ABB RobotStudio station: P4.rspag

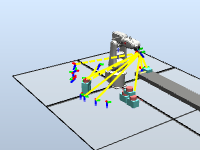
--- station ---
Station CPRClasificador (saved by RobotStudio 6.6.7701.1025)
Controller IRB_120_3kg_0.58m_1
  mechanical unit ROB_1: IRB120_3_58__01, 6 joints, base frame (0, 0, 0) mm
Layout (positions relative to the parent item):
  - Cinta [part]
  - Placa [part]
  - Disco [part]
  - CI_Ventosa [smart component]
      signals: DI ActivaVentosa, DO Vacuostato
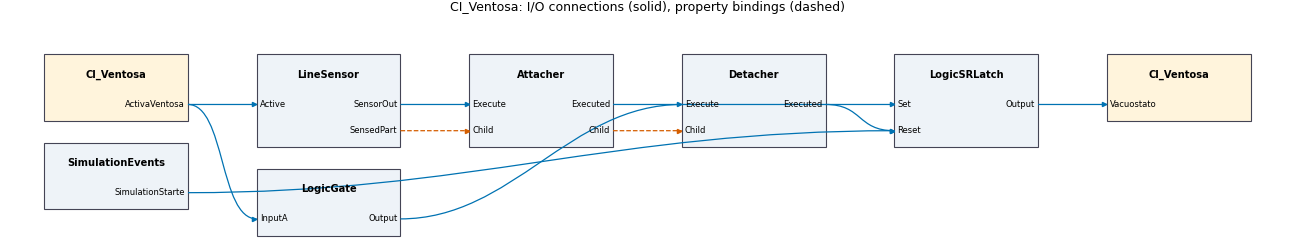
      connections:
        CI_Ventosa.ActivaVentosa -> LineSensor.Active
        LineSensor.SensorOut -> Attacher.Execute
        Attacher.Executed -> LogicSRLatch.Set
        Detacher.Executed -> LogicSRLatch.Reset
        CI_Ventosa.ActivaVentosa -> LogicGate.InputA
        LogicSRLatch.Output -> CI_Ventosa.Vacuostato
        SimulationEvents.SimulationStarted -> LogicSRLatch.Reset
        LogicGate.Output -> Detacher.Execute
        LineSensor.SensedPart => Attacher.Child
        Attacher.Child => Detacher.Child
    - LineSensor [smart component, from Components\LineSensor.rslib] at (364.35, 0, 594) mm, rotated rx 180 ry 60 rz 180 deg
        properties: Start=[0 0 0.049]; End=[0 0 0.061]; Radius=0.002; SensedPart=Disco_79; SensedPoint=[0.464333557128906 -0.180395202636719 0.20952131652832]
      - _sensorPart_ [part]
    - Attacher [smart component, from Components\Attacher.rslib]
        properties: Parent=MyNewTool; Flange=0; Child=Disco_79; Mount=false; Offset=[0 0 0]; Orientation=[0 0 0]
    - Detacher [smart component, from Components\Detacher.rslib]
        properties: Child=Disco_79; KeepPosition=true
    - LogicGate [smart component, from Components\LogicGate.rslib]
        properties: Operator=NOT; Delay=0
    - LogicSRLatch [smart component, from Components\LogicSRLatch.rslib]
    - SimulationEvents [smart component, from Components\SimulationEvents.rslib]
    - MyNewTool [mechanism] at (364.35, 0, 594) mm, rotated rx 180 ry 60 rz 180 deg
        TCP MyNewTool at (0, 0, 50) mm
        links: Cono
  - CI_Cinta [smart component]
      signals: DI ActivaSensores, DO SensorCinta1, DO SensorCinta2
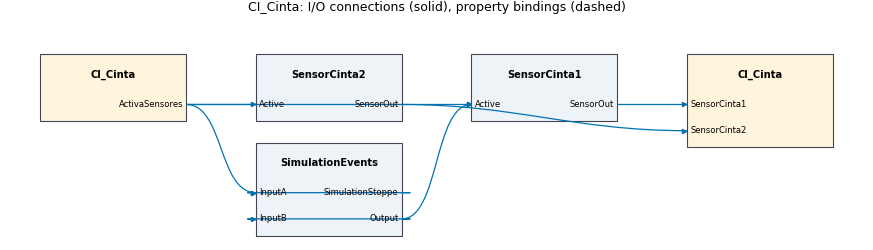
      connections:
        CI_Cinta.ActivaSensores -> SensorCinta2.Active
        SensorCinta1.SensorOut -> CI_Cinta.SensorCinta1
        SensorCinta2.SensorOut -> CI_Cinta.SensorCinta2
        SimulationEvents.SimulationStopped -> LogicGate_2.InputA
        LogicGate_2.Output -> LogicGate.InputB
        CI_Cinta.ActivaSensores -> LogicGate.InputA
        LogicGate.Output -> SensorCinta1.Active
        CI_Cinta.ActivaSensores -> SensorCinta1.Active
    - SensorCinta1 [smart component, from Components\LineSensor.rslib]
        properties: Start=[0.15 0.15 0.22]; End=[0.15 0.35 0.22]; Radius=0.002; SensedPart=Placa_91; SensedPoint=[0.15 0.25 0.22]
      - _sensorPart_ [part]
    - SensorCinta2 [smart component, from Components\LineSensor.rslib]
        properties: Start=[0.25 0.15 0.22]; End=[0.25 0.35 0.22]; Radius=0.002; SensedPart=Placa_91; SensedPoint=[0.25 0.25 0.22]
      - _sensorPart_ [part]
  - CI_Piezas [smart component]
      signals: DI Pieza, DI MotorCinta, DI Desencolar
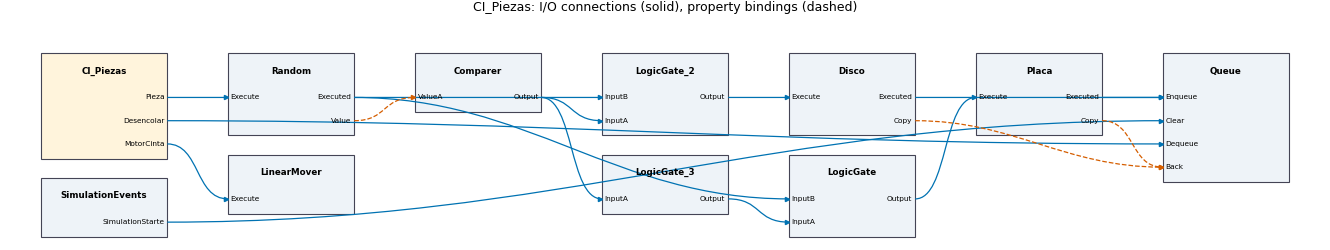
      connections:
        Random.Executed -> LogicGate_2.InputB
        Random.Executed -> LogicGate.InputB
        Comparer.Output -> LogicGate_2.InputA
        Comparer.Output -> LogicGate_3.InputA
        LogicGate_3.Output -> LogicGate.InputA
        LogicGate_2.Output -> Disco.Execute
        Disco.Executed -> Queue.Enqueue
        CI_Piezas.Pieza -> Random.Execute
        SimulationEvents.SimulationStarted -> Queue.Clear
        CI_Piezas.Desencolar -> Queue.Dequeue
        Placa.Executed -> Queue.Enqueue
        LogicGate.Output -> Placa.Execute
        CI_Piezas.MotorCinta -> LinearMover.Execute
        Random.Value => Comparer.ValueA
        Disco.Copy => Queue.Back
        Placa.Copy => Queue.Back
    - Disco [smart component, from Components\Source.rslib]
        properties: Source=Disco; Copy=Disco_171; Parent=(none); Position=[1.25 0.23 0.2]; Orientation=[0 0 0]; Transient=false; PhysicsBehavior=0
    - Random [smart component, from Components\Random.rslib]
        properties: Value=0.259914413215553; Min=0; Max=1
    - Comparer [smart component, from Components\Comparer.rslib]
        properties: ValueA=0.259914413215553; Operator=<=; ValueB=0.5
    - LogicGate [smart component, from Components\LogicGate.rslib]
        properties: Operator=AND; Delay=0
    - LogicGate_2 [smart component, from Components\LogicGate.rslib]
        properties: Operator=AND; Delay=0
    - LogicGate_3 [smart component, from Components\LogicGate.rslib]
        properties: Operator=NOT; Delay=0
    - LinearMover [smart component, from Components\LinearMover.rslib]
        properties: Object=Queue; Direction=[-1 0 0]; Speed=0.15; Reference=Global; ReferenceObject=(none)
    - SimulationEvents [smart component, from Components\SimulationEvents.rslib]
    - Queue [smart component, from Components\Queue.rslib]
        properties: Back=Disco_171; Front=Disco_171; Queue={b508ca64-a9cf-4086-8e21-28a4116258de}; NumberOfObjects=1
    - Placa [smart component, from Components\Source.rslib]
        properties: Source=Placa; Copy=Placa_170; Parent=(none); Position=[1.15 0.25 0.2]; Orientation=[0 0 0]; Transient=false; PhysicsBehavior=0
  - IRB120_3_58__01 [mechanism, from Robots\IRB120_3_58_G_01.rslib] at (0, 0, 0) mm; joint values [0, 0, 0, 0, 0.5236, 0] (rad or m)
  - Placa_75 [part] at (1150, 250, 200) mm
  - Placa_81 [part] at (1150, 250, 200) mm
  - Placa_83 [part] at (1150, 250, 200) mm
  - Placa_84 [part] at (1150, 250, 200) mm
  - Placa_85 [part] at (1150, 250, 200) mm
  - Placa_86 [part] at (1150, 250, 200) mm
  - Placa_88 [part] at (1150, 250, 200) mm
  - Placa_93 [part] at (1150, 250, 200) mm
  - Placa_94 [part] at (1150, 250, 200) mm
  - Placa_95 [part] at (1150, 250, 200) mm
  - Placa_97 [part] at (1150, 250, 200) mm
  - Placa_99 [part] at (1150, 250, 200) mm
  - Placa_101 [part] at (1150, 250, 200) mm
  - Placa_102 [part] at (1150, 250, 200) mm
  - Placa_103 [part] at (1150, 250, 200) mm
  - Placa_104 [part] at (1150, 250, 200) mm
  - Disco_105 [part] at (1250, 230, 200) mm
  - Disco_106 [part] at (1250, 230, 200) mm
  - Disco_107 [part] at (1250, 230, 200) mm
  - Disco_108 [part] at (1250, 230, 200) mm
  - Placa_110 [part] at (1150, 250, 200) mm
  - Placa_111 [part] at (1150, 250, 200) mm
  - Placa_113 [part] at (1150, 250, 200) mm
  - Disco_114 [part] at (1250, 230, 200) mm
  - Disco_115 [part] at (1250, 230, 200) mm
  - Placa_116 [part] at (1150, 250, 200) mm
  - Placa_117 [part] at (1150, 250, 200) mm
  - Disco_118 [part] at (1250, 230, 200) mm
  - Placa_119 [part] at (1150, 250, 200) mm
  - Disco_120 [part] at (1250, 230, 200) mm
  - Disco_121 [part] at (1250, 230, 200) mm
  - Disco_122 [part] at (1250, 230, 200) mm
  - Disco_123 [part] at (1250, 230, 200) mm
  - Placa_124 [part] at (1150, 250, 200) mm
  - Placa_125 [part] at (1150, 250, 200) mm
  - Placa_126 [part] at (1150, 250, 200) mm
  - Disco_127 [part] at (1250, 230, 200) mm
  - Placa_128 [part] at (1150, 250, 200) mm
  - Disco_129 [part] at (1250, 230, 200) mm
  - Placa_130 [part] at (1150, 250, 200) mm
  - Disco_131 [part] at (1250, 230, 200) mm
  - Placa_132 [part] at (1150, 250, 200) mm
  - Placa_133 [part] at (1150, 250, 200) mm
  - Placa_134 [part] at (1150, 250, 200) mm
  - Disco_135 [part] at (1250, 230, 200) mm
  - Disco_137 [part] at (1250, 230, 200) mm
  - Disco_138 [part] at (1250, 230, 200) mm
  - Disco_139 [part] at (1250, 230, 200) mm
  - Disco_140 [part] at (1250, 230, 200) mm
  - Disco_141 [part] at (1250, 230, 200) mm
  - Disco_142 [part] at (1250, 230, 200) mm
  - Placa_143 [part] at (1150, 250, 200) mm
  - Placa_144 [part] at (1150, 250, 200) mm
  - Disco_145 [part] at (1250, 230, 200) mm
  - Placa_146 [part] at (1150, 250, 200) mm
  - Disco_147 [part] at (1250, 230, 200) mm
  - Disco_148 [part] at (1250, 230, 200) mm
  - Placa_149 [part] at (1150, 250, 200) mm
  - Placa_150 [part] at (1150, 250, 200) mm
  - Disco_151 [part] at (1250, 230, 200) mm
  - Disco_152 [part] at (1250, 230, 200) mm
  - Placa_153 [part] at (1150, 250, 200) mm
  - Disco_154 [part] at (1250, 230, 200) mm
  - Placa_155 [part] at (1150, 250, 200) mm
  - Placa_156 [part] at (1150, 250, 200) mm
  - Disco_157 [part] at (1250, 230, 200) mm
  - Disco_158 [part] at (1250, 230, 200) mm
  - Placa_159 [part] at (1150, 250, 200) mm
  - Placa_161 [part] at (1150, 250, 200) mm
  - Placa_162 [part] at (1150, 250, 200) mm
  - Placa_163 [part] at (1150, 250, 200) mm
  - Disco_164 [part] at (1250, 230, 200) mm
  - Disco_165 [part] at (1250, 230, 200) mm
  - Placa_166 [part] at (1150, 250, 200) mm
  - Placa_167 [part] at (1150, 250, 200) mm
  - Disco_168 [part] at (1250, 230, 200) mm
  - Placa_169 [part] at (1150, 250, 200) mm
  - Disco_170 [part] at (1250, 230, 200) mm
  - Disco_171 [part] at (1250, 230, 200) mm
  - Disco_172 [part] at (1250, 230, 200) mm
  - Disco_173 [part] at (1250, 230, 200) mm
  - Disco_174 [part] at (1250, 230, 200) mm
  - Disco_175 [part] at (1250, 230, 200) mm
  - Disco_176 [part] at (1250, 230, 200) mm
  - Disco_177 [part] at (1250, 230, 200) mm
  - Disco_178 [part] at (1250, 230, 200) mm
  - Disco_179 [part] at (1250, 230, 200) mm
  - Disco_180 [part] at (1250, 230, 200) mm
  - Disco_181 [part] at (1250, 230, 200) mm
  - Placa_182 [part] at (1150, 250, 200) mm
  - Disco_183 [part] at (1250, 230, 200) mm
  - Disco_185 [part] at (1250, 230, 200) mm
  - Placa_186 [part] at (1150, 250, 200) mm
  - Disco_187 [part] at (1250, 230, 200) mm
  - Disco_188 [part] at (1250, 230, 200) mm
  - Placa_189 [part] at (1150, 250, 200) mm
  - Placa_190 [part] at (1150, 250, 200) mm
  - Placa_191 [part] at (1150, 250, 200) mm
  - Disco_192 [part] at (1250, 230, 200) mm
  - Disco_193 [part] at (1250, 230, 200) mm
  - Placa_194 [part] at (1150, 250, 200) mm
  - Disco_195 [part] at (1250, 230, 200) mm
  - Placa_196 [part] at (1150, 250, 200) mm
  - Placa_197 [part] at (1150, 250, 200) mm
  - Disco_198 [part] at (1250, 230, 200) mm
  - Disco_199 [part] at (1250, 230, 200) mm
  - Placa_200 [part] at (1150, 250, 200) mm
  - Placa_201 [part] at (1150, 250, 200) mm
  - Disco_202 [part] at (1250, 230, 200) mm
  - Placa_203 [part] at (1150, 250, 200) mm
  - Disco_204 [part] at (1250, 230, 200) mm
  - Disco_205 [part] at (1250, 230, 200) mm
  - Disco_206 [part] at (1250, 230, 200) mm
  - Disco_207 [part] at (1250, 230, 200) mm
  - Disco_209 [part] at (1250, 230, 200) mm
  - Placa_210 [part] at (1150, 250, 200) mm
  - Disco_211 [part] at (1250, 230, 200) mm
  - Disco_212 [part] at (1250, 230, 200) mm
  - Placa_213 [part] at (1150, 250, 200) mm
  - Placa_214 [part] at (1150, 250, 200) mm
  - Placa_215 [part] at (1150, 250, 200) mm
  - Disco_216 [part] at (1250, 230, 200) mm
  - Placa_217 [part] at (1150, 250, 200) mm
  - Disco_218 [part] at (1250, 230, 200) mm
  - Disco_219 [part] at (1250, 230, 200) mm
  - Disco_220 [part] at (1250, 230, 200) mm
  - Placa_221 [part] at (1150, 250, 200) mm
  - Placa_222 [part] at (1150, 250, 200) mm
  - Placa_223 [part] at (1150, 250, 200) mm
  - Disco_224 [part] at (1250, 230, 200) mm
  - Placa_225 [part] at (1150, 250, 200) mm
  - Disco_226 [part] at (1250, 230, 200) mm
  - Placa_227 [part] at (1150, 250, 200) mm
  - Placa_228 [part] at (1150, 250, 200) mm
  - Placa_229 [part] at (1150, 250, 200) mm
  - Placa_230 [part] at (1150, 250, 200) mm
  - Disco_231 [part] at (1250, 230, 200) mm
  - Placa_232 [part] at (1150, 250, 200) mm
  - Disco_233 [part] at (1250, 230, 200) mm
  - Placa_234 [part] at (1150, 250, 200) mm
  - Disco_235 [part] at (1250, 230, 200) mm
  - Disco_236 [part] at (1250, 230, 200) mm
  - Disco_237 [part] at (1250, 230, 200) mm
  - Placa_238 [part] at (1150, 250, 200) mm
  - Disco_239 [part] at (1250, 230, 200) mm
  - Disco_240 [part] at (1250, 230, 200) mm
  - Disco_241 [part] at (1250, 230, 200) mm
  - Placa_242 [part] at (1150, 250, 200) mm
  - Placa_243 [part] at (1150, 250, 200) mm
  - Placa_244 [part] at (1150, 250, 200) mm
  - Disco_245 [part] at (1250, 230, 200) mm
  - Placa_246 [part] at (1150, 250, 200) mm
  - Disco_247 [part] at (1250, 230, 200) mm
  - Placa_248 [part] at (1150, 250, 200) mm
  - Placa_249 [part] at (1150, 250, 200) mm
  - Disco_250 [part] at (1250, 230, 200) mm
  - Disco_251 [part] at (1250, 230, 200) mm
  - Disco_252 [part] at (1250, 230, 200) mm
  - Disco_253 [part] at (1250, 230, 200) mm
  - Placa_254 [part] at (1150, 250, 200) mm
  - Disco_255 [part] at (1250, 230, 200) mm
  - Placa_256 [part] at (1150, 250, 200) mm
  - Disco_257 [part] at (1250, 230, 200) mm
  - Placa_258 [part] at (1150, 250, 200) mm
  - Placa_259 [part] at (1150, 250, 200) mm
  - Disco_260 [part] at (1250, 230, 200) mm
  - Disco_261 [part] at (1250, 230, 200) mm
  - Placa_262 [part] at (1150, 250, 200) mm
  - Placa_263 [part] at (1150, 250, 200) mm
  - Placa_264 [part] at (1150, 250, 200) mm
  - Disco_265 [part] at (1250, 230, 200) mm
  - Disco_266 [part] at (1250, 230, 200) mm
  - Placa_267 [part] at (1150, 250, 200) mm
  - Disco_268 [part] at (1250, 230, 200) mm
  - Disco_269 [part] at (1250, 230, 200) mm
  - Disco_270 [part] at (1250, 230, 200) mm
  - Placa_271 [part] at (1150, 250, 200) mm
  - Placa_272 [part] at (1150, 250, 200) mm
  - Disco_273 [part] at (1250, 230, 200) mm
  - Disco_274 [part] at (1250, 230, 200) mm
  - Placa_275 [part] at (1150, 250, 200) mm
  - Placa_276 [part] at (1150, 250, 200) mm
  - Disco_277 [part] at (1250, 230, 200) mm
  - Placa_278 [part] at (1150, 250, 200) mm
  - Placa_279 [part] at (1150, 250, 200) mm
  - Disco_280 [part] at (1250, 230, 200) mm
  - Placa_281 [part] at (1150, 250, 200) mm
  - Disco_282 [part] at (1250, 230, 200) mm
  - Placa_283 [part] at (1150, 250, 200) mm
  - Disco_284 [part] at (1250, 230, 200) mm
  - Disco_285 [part] at (1250, 230, 200) mm
  - Disco_286 [part] at (1250, 230, 200) mm
  - Placa_287 [part] at (1150, 250, 200) mm
  - Disco_288 [part] at (1250, 230, 200) mm
  - Disco_289 [part] at (1250, 230, 200) mm
  - Disco_290 [part] at (1250, 230, 200) mm
  - Placa_291 [part] at (1150, 250, 200) mm
  - Placa_292 [part] at (1150, 250, 200) mm
  - Placa_293 [part] at (1150, 250, 200) mm
  - Placa_294 [part] at (1150, 250, 200) mm
  - Placa_295 [part] at (1150, 250, 200) mm
  - Placa_296 [part] at (1150, 250, 200) mm
  - Placa_297 [part] at (1150, 250, 200) mm
  - Placa_298 [part] at (1150, 250, 200) mm
  - Disco_299 [part] at (1250, 230, 200) mm
  - Placa_300 [part] at (1150, 250, 200) mm
  - Placa_301 [part] at (1150, 250, 200) mm
  - Disco_302 [part] at (1250, 230, 200) mm
  - Disco_303 [part] at (1250, 230, 200) mm
  - Placa_304 [part] at (1150, 250, 200) mm
  - Placa_305 [part] at (1150, 250, 200) mm
  - Disco_306 [part] at (1250, 230, 200) mm
  - Disco_307 [part] at (1250, 230, 200) mm
  - Placa_308 [part] at (1150, 250, 200) mm
  - Placa_309 [part] at (1150, 250, 200) mm
  - Disco_310 [part] at (1250, 230, 200) mm
  - Placa_311 [part] at (1150, 250, 200) mm
  - Placa_312 [part] at (1150, 250, 200) mm
  - Placa_313 [part] at (1150, 250, 200) mm
  - Placa_314 [part] at (1150, 250, 200) mm
  - Placa_315 [part] at (1150, 250, 200) mm
  - Placa_316 [part] at (1150, 250, 200) mm
  - Disco_317 [part] at (1250, 230, 200) mm
  - Placa_318 [part] at (1150, 250, 200) mm
  - Disco_319 [part] at (1250, 230, 200) mm
  - Disco_320 [part] at (1250, 230, 200) mm
  - Placa_321 [part] at (1150, 250, 200) mm
  - Placa_322 [part] at (1150, 250, 200) mm
  - Placa_323 [part] at (1150, 250, 200) mm
  - Disco_324 [part] at (1250, 230, 200) mm
  - Disco_325 [part] at (1250, 230, 200) mm
  - Disco_326 [part] at (1250, 230, 200) mm
  - Placa_327 [part] at (1150, 250, 200) mm
  - Disco_328 [part] at (1250, 230, 200) mm
  - Disco_329 [part] at (1250, 230, 200) mm
  - Disco_330 [part] at (1250, 230, 200) mm
  - Disco_331 [part] at (1250, 230, 200) mm
  - Disco_332 [part] at (1250, 230, 200) mm
  - Disco_333 [part] at (1250, 230, 200) mm
  - Placa_334 [part] at (1150, 250, 200) mm
  - Disco_335 [part] at (1250, 230, 200) mm
  - Placa_336 [part] at (1150, 250, 200) mm
  - Disco_337 [part] at (1250, 230, 200) mm
  - Placa_338 [part] at (1150, 250, 200) mm
  - Placa_339 [part] at (1150, 250, 200) mm
  - Disco_340 [part] at (1250, 230, 200) mm
  - Placa_341 [part] at (1150, 250, 200) mm
  - Disco_342 [part] at (1250, 230, 200) mm
  - Disco_343 [part] at (1250, 230, 200) mm
  - Disco_344 [part] at (1250, 230, 200) mm
  - Disco_345 [part] at (1250, 230, 200) mm
  - Disco_346 [part] at (1250, 230, 200) mm
  - Placa_347 [part] at (1150, 250, 200) mm
  - Disco_348 [part] at (1250, 230, 200) mm
  - Disco_349 [part] at (1250, 230, 200) mm
  - Disco_350 [part] at (1250, 230, 200) mm
  - Placa_351 [part] at (1150, 250, 200) mm
  - Disco_7 [part] at (1250, 230, 200) mm
  - Disco_8 [part] at (1250, 230, 200) mm
  - Disco_9 [part] at (1250, 230, 200) mm
  - Disco_10 [part] at (1250, 230, 200) mm
  - Disco_11 [part] at (1250, 230, 200) mm
  - Disco_12 [part] at (1250, 230, 200) mm
  - Disco_13 [part] at (1250, 230, 200) mm
  - Disco_14 [part] at (1250, 230, 200) mm
  - Placa_15 [part] at (1150, 250, 200) mm
  - Placa_16 [part] at (1150, 250, 200) mm
  - Placa_17 [part] at (1150, 250, 200) mm
  - Disco_18 [part] at (1250, 230, 200) mm
  - Disco_20 [part] at (1250, 230, 200) mm
  - Placa_21 [part] at (1150, 250, 200) mm
  - Placa_22 [part] at (1150, 250, 200) mm
  - Placa_23 [part] at (1150, 250, 200) mm
  - Disco_24 [part] at (1250, 230, 200) mm
  - Disco_25 [part] at (1250, 230, 200) mm
  - Placa_26 [part] at (1150, 250, 200) mm
  - Placa_27 [part] at (1150, 250, 200) mm
  - Disco_28 [part] at (1250, 230, 200) mm
  - Disco_29 [part] at (1250, 230, 200) mm
  - Placa_30 [part] at (1150, 250, 200) mm
  - Placa_31 [part] at (1150, 250, 200) mm
  - Placa_32 [part] at (1150, 250, 200) mm
  - Disco_33 [part] at (1250, 230, 200) mm
  - Disco_34 [part] at (1250, 230, 200) mm
  - Placa_35 [part] at (1150, 250, 200) mm
  - Placa_36 [part] at (1150, 250, 200) mm
  - Placa_37 [part] at (1150, 250, 200) mm
  - Disco_38 [part] at (1250, 230, 200) mm
  - Disco_39 [part] at (1250, 230, 200) mm
  - Placa_40 [part] at (1150, 250, 200) mm
  - Placa_41 [part] at (1150, 250, 200) mm
  - Placa_42 [part] at (1150, 250, 200) mm
  - Placa_44 [part] at (1150, 250, 200) mm
  - Placa_45 [part] at (1150, 250, 200) mm
  - Disco_46 [part] at (1250, 230, 200) mm
  - Placa_47 [part] at (1150, 250, 200) mm
  - Disco_48 [part] at (1250, 230, 200) mm
  - Placa_49 [part] at (1150, 250, 200) mm
  - Placa_50 [part] at (1150, 250, 200) mm
  - Placa_51 [part] at (1150, 250, 200) mm
  - Disco_52 [part] at (1250, 230, 200) mm
  - Disco_53 [part] at (1250, 230, 200) mm
  - Placa_54 [part] at (1150, 250, 200) mm
  - Placa_55 [part] at (1150, 250, 200) mm
  - Placa_56 [part] at (1150, 250, 200) mm
  - Disco_57 [part] at (1250, 230, 200) mm
  - Disco_58 [part] at (1250, 230, 200) mm
  - Placa_59 [part] at (1150, 250, 200) mm
  - Disco_60 [part] at (1250, 230, 200) mm
  - Disco_61 [part] at (1250, 230, 200) mm
  - Placa_62 [part] at (1150, 250, 200) mm
  - Disco_63 [part] at (1250, 230, 200) mm
  - Disco_64 [part] at (1250, 230, 200) mm
  - Placa_65 [part] at (1150, 250, 200) mm
  - Placa_66 [part] at (1150, 250, 200) mm
  - Disco_68 [part] at (1250, 230, 200) mm
  - Disco_69 [part] at (1250, 230, 200) mm
  - Placa_70 [part] at (1150, 250, 200) mm
  - Disco_71 [part] at (1250, 230, 200) mm
  - Disco_72 [part] at (1250, 230, 200) mm
  - Disco_73 [part] at (1250, 230, 200) mm
  - Disco_74 [part] at (1250, 230, 200) mm
  - Placa_75 [part] at (1150, 250, 200) mm
  - Placa_76 [part] at (1150, 250, 200) mm
  - Disco_77 [part] at (1250, 230, 200) mm
  - Disco_78 [part] at (1250, 230, 200) mm
  - Placa_79 [part] at (1150, 250, 200) mm
  - Placa_80 [part] at (1150, 250, 200) mm
  - Placa_81 [part] at (1150, 250, 200) mm
  - Placa_82 [part] at (1150, 250, 200) mm
  - Disco_83 [part] at (1250, 230, 200) mm
  - Disco_84 [part] at (1250, 230, 200) mm
  - Disco_85 [part] at (1250, 230, 200) mm
  - Placa_86 [part] at (1150, 250, 200) mm
  - Disco_87 [part] at (1250, 230, 200) mm
  - Disco_88 [part] at (1250, 230, 200) mm
  - Disco_89 [part] at (1250, 230, 200) mm
  - Disco_90 [part] at (1250, 230, 200) mm
  - Placa_91 [part] at (1150, 250, 200) mm
  - Disco_92 [part] at (1250, 230, 200) mm
  - Placa_93 [part] at (1150, 250, 200) mm
  - Disco_94 [part] at (1250, 230, 200) mm
  - Placa_95 [part] at (1150, 250, 200) mm
  - Placa_96 [part] at (1150, 250, 200) mm
  - Placa_97 [part] at (1150, 250, 200) mm
  - Disco_98 [part] at (1250, 230, 200) mm
  - Placa_99 [part] at (1150, 250, 200) mm
  - Placa_100 [part] at (1150, 250, 200) mm
  - Disco_101 [part] at (1250, 230, 200) mm
  - Placa_102 [part] at (1150, 250, 200) mm
  - Placa_103 [part] at (1150, 250, 200) mm
  - Disco_104 [part] at (1250, 230, 200) mm
  - Disco_105 [part] at (1250, 230, 200) mm
  - Disco_106 [part] at (1250, 230, 200) mm
  - Disco_107 [part] at (1250, 230, 200) mm
  - Disco_108 [part] at (1250, 230, 200) mm
  - Disco_109 [part] at (1250, 230, 200) mm
  - Placa_110 [part] at (1150, 250, 200) mm
  - Placa_111 [part] at (1150, 250, 200) mm
  - Placa_112 [part] at (1150, 250, 200) mm
  - Disco_113 [part] at (1250, 230, 200) mm
  - Placa_114 [part] at (1150, 250, 200) mm
  - Disco_115 [part] at (1250, 230, 200) mm
  - Disco_116 [part] at (1250, 230, 200) mm
  - Placa_117 [part] at (1150, 250, 200) mm
  - Placa_118 [part] at (1150, 250, 200) mm
  - Disco_119 [part] at (1250, 230, 200) mm
  - Disco_120 [part] at (1250, 230, 200) mm
  - Disco_121 [part] at (1250, 230, 200) mm
  - Placa_122 [part] at (1150, 250, 200) mm
  - Placa_123 [part] at (1150, 250, 200) mm
  - Disco_124 [part] at (1250, 230, 200) mm
  - Placa_125 [part] at (1150, 250, 200) mm
  - Disco_126 [part] at (1250, 230, 200) mm
  - Placa_127 [part] at (1150, 250, 200) mm
  - Placa_128 [part] at (1150, 250, 200) mm
  - Disco_129 [part] at (1250, 230, 200) mm
  - Placa_130 [part] at (1150, 250, 200) mm
  - Disco_131 [part] at (1250, 230, 200) mm
  - Placa_132 [part] at (1150, 250, 200) mm
  - Disco_133 [part] at (1250, 230, 200) mm
  - Disco_134 [part] at (1250, 230, 200) mm
  - Placa_135 [part] at (1150, 250, 200) mm
  - Placa_136 [part] at (1150, 250, 200) mm
  - Disco_137 [part] at (1250, 230, 200) mm
  - Disco_138 [part] at (1250, 230, 200) mm
  - Disco_139 [part] at (1250, 230, 200) mm
  - Placa_140 [part] at (1150, 250, 200) mm
  - Disco_141 [part] at (1250, 230, 200) mm
  - Disco_142 [part] at (1250, 230, 200) mm
  - Placa_143 [part] at (1150, 250, 200) mm
  - Placa_144 [part] at (1150, 250, 200) mm
  - Placa_145 [part] at (1150, 250, 200) mm
  - Placa_146 [part] at (1150, 250, 200) mm
  - Disco_147 [part] at (1250, 230, 200) mm
  - Placa_148 [part] at (1150, 250, 200) mm
  - Placa_149 [part] at (1150, 250, 200) mm
  - Placa_150 [part] at (1150, 250, 200) mm
  - Disco_151 [part] at (1250, 230, 200) mm
  - Disco_152 [part] at (1250, 230, 200) mm
  - Disco_153 [part] at (1250, 230, 200) mm
  - Disco_154 [part] at (1250, 230, 200) mm
  - Disco_155 [part] at (1250, 230, 200) mm
  - Disco_156 [part] at (1250, 230, 200) mm
  - Disco_157 [part] at (1250, 230, 200) mm
  - Disco_158 [part] at (1250, 230, 200) mm
  - Disco_159 [part] at (1250, 230, 200) mm
  - Disco_160 [part] at (1250, 230, 200) mm
  - Placa_161 [part] at (1150, 250, 200) mm
  - Placa_163 [part] at (1150, 250, 200) mm
  - Disco_164 [part] at (1250, 230, 200) mm
  - Placa_165 [part] at (1150, 250, 200) mm
  - Placa_166 [part] at (1150, 250, 200) mm
  - Disco_167 [part] at (1250, 230, 200) mm
  - Disco_168 [part] at (1250, 230, 200) mm
  - Disco_169 [part] at (1250, 230, 200) mm
  - Placa_170 [part] at (1150, 250, 200) mm
  - Disco_171 [part] at (1250, 230, 200) mm
  - Disco_172 [part] at (1250, 230, 200) mm
  - Placa_173 [part] at (1150, 250, 200) mm
  - Disco_174 [part] at (1250, 230, 200) mm
  - Placa_175 [part] at (1150, 250, 200) mm
  - Placa_176 [part] at (1150, 250, 200) mm
  - Disco_177 [part] at (1250, 230, 200) mm
  - Disco_178 [part] at (1250, 230, 200) mm
  - Placa_179 [part] at (1150, 250, 200) mm
  - Placa_180 [part] at (1150, 250, 200) mm
  - Placa_181 [part] at (1150, 250, 200) mm
  - Placa_182 [part] at (1150, 250, 200) mm
  - Disco_183 [part] at (1250, 230, 200) mm
  - Placa_184 [part] at (1150, 250, 200) mm
  - Placa_185 [part] at (1150, 250, 200) mm
  - Disco_186 [part] at (1250, 230, 200) mm
  - Disco_187 [part] at (1250, 230, 200) mm
  - Disco_188 [part] at (1250, 230, 200) mm
  - Placa_189 [part] at (1150, 250, 200) mm
  - Disco_190 [part] at (1250, 230, 200) mm
  - Disco_191 [part] at (1250, 230, 200) mm
  - Placa_192 [part] at (1150, 250, 200) mm
  - Disco_193 [part] at (1250, 230, 200) mm
  - Placa_194 [part] at (1150, 250, 200) mm
  - Disco_195 [part] at (1250, 230, 200) mm
  - Disco_196 [part] at (1250, 230, 200) mm
  - Placa_197 [part] at (1150, 250, 200) mm
  - Disco_198 [part] at (1250, 230, 200) mm
  - Disco_199 [part] at (1250, 230, 200) mm
  - Placa_200 [part] at (1150, 250, 200) mm
  - Disco_201 [part] at (1250, 230, 200) mm
  - Disco_202 [part] at (1250, 230, 200) mm
  - Placa_203 [part] at (1150, 250, 200) mm
  - Placa_204 [part] at (1150, 250, 200) mm
  - Placa_205 [part] at (1150, 250, 200) mm
  - Placa_206 [part] at (1150, 250, 200) mm
  - Disco_207 [part] at (1250, 230, 200) mm
  - Placa_208 [part] at (1150, 250, 200) mm
  - Disco_209 [part] at (1250, 230, 200) mm
  - Placa_219 [part] at (1150, 250, 200) mm
  - Disco_220 [part] at (1250, 230, 200) mm
  - Disco_221 [part] at (1250, 230, 200) mm
  - Disco_222 [part] at (1250, 230, 200) mm
  - Disco_223 [part] at (1250, 230, 200) mm
  - Disco_224 [part] at (1250, 230, 200) mm
  - Placa_225 [part] at (1150, 250, 200) mm
  - Disco_226 [part] at (1250, 230, 200) mm
  - Disco_227 [part] at (1250, 230, 200) mm
  - Placa_228 [part] at (1150, 250, 200) mm
  - Disco_229 [part] at (1250, 230, 200) mm
  - Disco_231 [part] at (1250, 230, 200) mm
  - Placa_232 [part] at (1150, 250, 200) mm
  - Disco_233 [part] at (1250, 230, 200) mm
  - Placa_234 [part] at (1150, 250, 200) mm
  - Placa_235 [part] at (1150, 250, 200) mm
  - Placa_236 [part] at (1150, 250, 200) mm
  - Disco_237 [part] at (1250, 230, 200) mm
  - Placa_238 [part] at (1150, 250, 200) mm
  - Disco_239 [part] at (1250, 230, 200) mm
  - Placa_240 [part] at (1150, 250, 200) mm
  - Placa_241 [part] at (1150, 250, 200) mm
  - Placa_242 [part] at (1150, 250, 200) mm
  - Placa_243 [part] at (1150, 250, 200) mm
  - Disco_244 [part] at (1250, 230, 200) mm
  - Disco_245 [part] at (1250, 230, 200) mm
  - Disco_246 [part] at (1250, 230, 200) mm
  - Placa_247 [part] at (1150, 250, 200) mm
  - Placa_248 [part] at (1150, 250, 200) mm
  - Placa_249 [part] at (1150, 250, 200) mm
  - Disco_250 [part] at (1250, 230, 200) mm
  - Placa_251 [part] at (1150, 250, 200) mm
  - Placa_252 [part] at (1150, 250, 200) mm
  - Placa_253 [part] at (1150, 250, 200) mm
  - Disco_255 [part] at (1250, 230, 200) mm
  - Disco_256 [part] at (1250, 230, 200) mm
  - Placa_257 [part] at (1150, 250, 200) mm
  - Placa_258 [part] at (1150, 250, 200) mm
  - Disco_259 [part] at (1250, 230, 200) mm
  - Disco_260 [part] at (1250, 230, 200) mm
  - Placa_261 [part] at (1150, 250, 200) mm
  - Placa_262 [part] at (1150, 250, 200) mm
  - Placa_263 [part] at (1150, 250, 200) mm
  - Placa_264 [part] at (1150, 250, 200) mm
  - Disco_265 [part] at (1250, 230, 200) mm
  - Disco_266 [part] at (1250, 230, 200) mm
  - Disco_267 [part] at (1250, 230, 200) mm
  - Disco_268 [part] at (1250, 230, 200) mm
  - Placa_269 [part] at (1150, 250, 200) mm
  - Placa_270 [part] at (1150, 250, 200) mm
  - Placa_271 [part] at (1150, 250, 200) mm
  - Placa_272 [part] at (1150, 250, 200) mm
  - Placa_273 [part] at (1150, 250, 200) mm
  - Placa_274 [part] at (1150, 250, 200) mm
  - Placa_275 [part] at (1150, 250, 200) mm
  - Placa_276 [part] at (1150, 250, 200) mm
  - Disco_277 [part] at (1250, 230, 200) mm
  - Placa_279 [part] at (1150, 250, 200) mm
  - Disco_280 [part] at (1250, 230, 200) mm
  - Placa_281 [part] at (1150, 250, 200) mm
  - Disco_282 [part] at (1250, 230, 200) mm
  - Disco_283 [part] at (1250, 230, 200) mm
  - Disco_284 [part] at (1250, 230, 200) mm
  - Placa_285 [part] at (1150, 250, 200) mm
  - Placa_286 [part] at (1150, 250, 200) mm
  - Disco_287 [part] at (1250, 230, 200) mm
  - Disco_288 [part] at (1250, 230, 200) mm
  - Placa_289 [part] at (1150, 250, 200) mm
  - Disco_290 [part] at (1250, 230, 200) mm
  - Disco_291 [part] at (1250, 230, 200) mm
  - Placa_292 [part] at (1150, 250, 200) mm
  - Placa_293 [part] at (1150, 250, 200) mm
  - Placa_294 [part] at (1150, 250, 200) mm
  - Placa_295 [part] at (1150, 250, 200) mm
  - Disco_296 [part] at (1250, 230, 200) mm
  - Placa_297 [part] at (1150, 250, 200) mm
  - Placa_298 [part] at (1150, 250, 200) mm
  - Placa_299 [part] at (1150, 250, 200) mm
  - Placa_300 [part] at (1150, 250, 200) mm
  - Disco_301 [part] at (1250, 230, 200) mm
  - Disco_303 [part] at (1250, 230, 200) mm
  - Disco_304 [part] at (1250, 230, 200) mm
  - Disco_305 [part] at (1250, 230, 200) mm
  - Placa_306 [part] at (1150, 250, 200) mm
  - Placa_307 [part] at (1150, 250, 200) mm
  - Placa_308 [part] at (1150, 250, 200) mm
  - Disco_309 [part] at (1250, 230, 200) mm
  - Disco_310 [part] at (1250, 230, 200) mm
  - Placa_311 [part] at (1150, 250, 200) mm
  - Placa_312 [part] at (1150, 250, 200) mm
  - Placa_313 [part] at (1150, 250, 200) mm
  - Placa_314 [part] at (1150, 250, 200) mm
  - Placa_315 [part] at (1150, 250, 200) mm
  - Placa_316 [part] at (1150, 250, 200) mm
  - Placa_317 [part] at (1150, 250, 200) mm
  - Disco_318 [part] at (1250, 230, 200) mm
  - Disco_319 [part] at (1250, 230, 200) mm
  - Placa_320 [part] at (1150, 250, 200) mm
  - Placa_321 [part] at (1150, 250, 200) mm
  - Placa_322 [part] at (1150, 250, 200) mm
  - Placa_323 [part] at (1150, 250, 200) mm
  - Disco_324 [part] at (1250, 230, 200) mm
  - Placa_325 [part] at (1150, 250, 200) mm
  - Disco_326 [part] at (1250, 230, 200) mm
  - Disco_338 [part] at (1250, 230, 200) mm
  - Placa_339 [part] at (1150, 250, 200) mm
  - Placa_340 [part] at (1150, 250, 200) mm
  - Placa_341 [part] at (1150, 250, 200) mm
  - Placa_342 [part] at (1150, 250, 200) mm
  - Disco_343 [part] at (1250, 230, 200) mm
  - Disco_344 [part] at (1250, 230, 200) mm
  - Placa_345 [part] at (1150, 250, 200) mm
  - Disco_346 [part] at (1250, 230, 200) mm
  - Disco_347 [part] at (1250, 230, 200) mm
  - Placa_348 [part] at (1150, 250, 200) mm
  - Placa_349 [part] at (1150, 250, 200) mm
  - Disco_350 [part] at (1250, 230, 200) mm
  - Disco_351 [part] at (1250, 230, 200) mm
  - Disco_352 [part] at (1250, 230, 200) mm
  - Placa_353 [part] at (1150, 250, 200) mm
  - Disco_354 [part] at (1250, 230, 200) mm
  - Disco_355 [part] at (1250, 230, 200) mm
  - Disco_356 [part] at (1250, 230, 200) mm
  - Disco_357 [part] at (1250, 230, 200) mm
  - Placa_358 [part] at (1150, 250, 200) mm
  - Placa_359 [part] at (1150, 250, 200) mm
  - Disco_360 [part] at (1250, 230, 200) mm
  - Placa_362 [part] at (1150, 250, 200) mm
  - Placa_363 [part] at (1150, 250, 200) mm
  - Disco_364 [part] at (1250, 230, 200) mm
  - Disco_365 [part] at (1250, 230, 200) mm
  - Disco_366 [part] at (1250, 230, 200) mm
  - Disco_367 [part] at (1250, 230, 200) mm
  - Placa_368 [part] at (1150, 250, 200) mm
  - Placa_369 [part] at (1150, 250, 200) mm
  - Disco_370 [part] at (1250, 230, 200) mm
  - Disco_371 [part] at (1250, 230, 200) mm
  - Disco_372 [part] at (1250, 230, 200) mm
  - Placa_373 [part] at (1150, 250, 200) mm
  - Disco_374 [part] at (1250, 230, 200) mm
  - Placa_375 [part] at (1150, 250, 200) mm
  - Disco_376 [part] at (1250, 230, 200) mm
  - Disco_377 [part] at (1250, 230, 200) mm
  - Disco_378 [part] at (1250, 230, 200) mm
  - Placa_379 [part] at (1150, 250, 200) mm
  - Disco_380 [part] at (1250, 230, 200) mm
  - Placa_381 [part] at (1150, 250, 200) mm
  - Placa_382 [part] at (1150, 250, 200) mm
  - Disco_383 [part] at (1250, 230, 200) mm
  - Placa_384 [part] at (1150, 250, 200) mm
  - Placa_386 [part] at (1150, 250, 200) mm
  - Placa_387 [part] at (1150, 250, 200) mm
  - Disco_388 [part] at (1250, 230, 200) mm
  - Placa_389 [part] at (1150, 250, 200) mm
  - Placa_390 [part] at (1150, 250, 200) mm
  - Placa_391 [part] at (1150, 250, 200) mm
  - Placa_392 [part] at (1150, 250, 200) mm
  - Placa_393 [part] at (1150, 250, 200) mm
  - Placa_394 [part] at (1150, 250, 200) mm
  - Placa_395 [part] at (1150, 250, 200) mm
  - Disco_396 [part] at (1250, 230, 200) mm
  - Disco_397 [part] at (1250, 230, 200) mm
  - Placa_398 [part] at (1150, 250, 200) mm
  - Disco_399 [part] at (1250, 230, 200) mm
  - Disco_400 [part] at (1250, 230, 200) mm
  - Placa_401 [part] at (1150, 250, 200) mm
  - Disco_402 [part] at (1250, 230, 200) mm
  - Disco_403 [part] at (1250, 230, 200) mm
  - Placa_404 [part] at (1150, 250, 200) mm
  - Disco_405 [part] at (1250, 230, 200) mm
  - Placa_406 [part] at (1150, 250, 200) mm
  - Placa_407 [part] at (1150, 250, 200) mm
  - Disco_408 [part] at (1250, 230, 200) mm
  - Disco_410 [part] at (1250, 230, 200) mm
  - Disco_411 [part] at (1250, 230, 200) mm
  - Placa_412 [part] at (1150, 250, 200) mm
  - Placa_413 [part] at (1150, 250, 200) mm
  - Disco_414 [part] at (1250, 230, 200) mm
  - Disco_415 [part] at (1250, 230, 200) mm
  - Placa_416 [part] at (1150, 250, 200) mm
  - Disco_417 [part] at (1250, 230, 200) mm
  - Disco_418 [part] at (1250, 230, 200) mm
  - Disco_419 [part] at (1250, 230, 200) mm
  - Placa_420 [part] at (1150, 250, 200) mm
  - Disco_421 [part] at (1250, 230, 200) mm
  - Disco_422 [part] at (1250, 230, 200) mm
  - Disco_423 [part] at (1250, 230, 200) mm
  - Placa_424 [part] at (1150, 250, 200) mm
  - Disco_425 [part] at (1250, 230, 200) mm
  - Placa_426 [part] at (1150, 250, 200) mm
  - Placa_427 [part] at (1150, 250, 200) mm
  - Disco_428 [part] at (1250, 230, 200) mm
  - Placa_429 [part] at (1150, 250, 200) mm
  - Placa_430 [part] at (1150, 250, 200) mm
  - Placa_431 [part] at (1150, 250, 200) mm
  - Disco_432 [part] at (1250, 230, 200) mm
  - Disco_434 [part] at (1250, 230, 200) mm
  - Disco_435 [part] at (1250, 230, 200) mm
  - Placa_436 [part] at (1150, 250, 200) mm
  - Disco_437 [part] at (1250, 230, 200) mm
  - Disco_438 [part] at (1250, 230, 200) mm
  - Disco_439 [part] at (1250, 230, 200) mm
  - Disco_440 [part] at (1250, 230, 200) mm
  - Placa_441 [part] at (1150, 250, 200) mm
  - Disco_442 [part] at (1250, 230, 200) mm
  - Placa_443 [part] at (1150, 250, 200) mm
  - Placa_444 [part] at (1150, 250, 200) mm
  - Placa_445 [part] at (1150, 250, 200) mm
  - Placa_446 [part] at (1150, 250, 200) mm
  - Placa_447 [part] at (1150, 250, 200) mm
  - Disco_448 [part] at (1250, 230, 200) mm
  - Disco_449 [part] at (1250, 230, 200) mm
  - Placa_450 [part] at (1150, 250, 200) mm
  - Placa_451 [part] at (1150, 250, 200) mm
  - Disco_452 [part] at (1250, 230, 200) mm
  - Placa_453 [part] at (1150, 250, 200) mm
  - Placa_454 [part] at (1150, 250, 200) mm
  - Disco_455 [part] at (1250, 230, 200) mm
  - Placa_456 [part] at (1150, 250, 200) mm
  - Disco_457 [part] at (1250, 230, 200) mm
  - Placa_458 [part] at (1150, 250, 200) mm
  - Disco_459 [part] at (1250, 230, 200) mm
  - Placa_460 [part] at (1150, 250, 200) mm
  - Disco_461 [part] at (1250, 230, 200) mm
  - Placa_462 [part] at (1150, 250, 200) mm
  - Placa_463 [part] at (1150, 250, 200) mm
  - Disco_464 [part] at (1250, 230, 200) mm
  - Disco_465 [part] at (1250, 230, 200) mm
  - Placa_466 [part] at (1150, 250, 200) mm
  - Placa_467 [part] at (1150, 250, 200) mm
  - Disco_468 [part] at (1250, 230, 200) mm
  - Disco_469 [part] at (1250, 230, 200) mm
  - Placa_470 [part] at (1150, 250, 200) mm
  - Disco_471 [part] at (1250, 230, 200) mm
  - Placa_472 [part] at (1150, 250, 200) mm
  - Placa_473 [part] at (1150, 250, 200) mm
  - Disco_474 [part] at (1250, 230, 200) mm
  - Placa_475 [part] at (1150, 250, 200) mm
  - Placa_476 [part] at (1150, 250, 200) mm
  - Placa_477 [part] at (1150, 250, 200) mm
  - Disco_478 [part] at (1250, 230, 200) mm
  - Disco_479 [part] at (1250, 230, 200) mm
  - Placa_480 [part] at (1150, 250, 200) mm
  - Placa_481 [part] at (1150, 250, 200) mm
  - Placa_482 [part] at (1150, 250, 200) mm
  - Placa_483 [part] at (1150, 250, 200) mm
  - Placa_484 [part] at (1150, 250, 200) mm
  - Placa_485 [part] at (1150, 250, 200) mm
  - Placa_486 [part] at (1150, 250, 200) mm
  - Placa_487 [part] at (1150, 250, 200) mm
  - Placa_488 [part] at (1150, 250, 200) mm
  - Disco_489 [part] at (1250, 230, 200) mm
  - Placa_490 [part] at (1150, 250, 200) mm
  - Disco_491 [part] at (1250, 230, 200) mm
  - Placa_492 [part] at (1150, 250, 200) mm
  - Placa_493 [part] at (1150, 250, 200) mm
  - Placa_494 [part] at (1150, 250, 200) mm
  - Disco_495 [part] at (1250, 230, 200) mm
  - Disco_496 [part] at (1250, 230, 200) mm
  - Placa_497 [part] at (1150, 250, 200) mm
  - Disco_498 [part] at (1250, 230, 200) mm
  - Disco_499 [part] at (1250, 230, 200) mm
  - Placa_500 [part] at (1150, 250, 200) mm
  - Disco_501 [part] at (1250, 230, 200) mm
  - Placa_502 [part] at (1150, 250, 200) mm
  - Placa_503 [part] at (1150, 250, 200) mm
  - Disco_504 [part] at (1250, 230, 200) mm
  - Placa_505 [part] at (1150, 250, 200) mm
  - Disco_506 [part] at (1250, 230, 200) mm
  - Placa_507 [part] at (1150, 250, 200) mm
  - Placa_508 [part] at (1150, 250, 200) mm
  - Placa_509 [part] at (1150, 250, 200) mm
  - Disco_510 [part] at (1250, 230, 200) mm
  - Disco_511 [part] at (1250, 230, 200) mm
  - Placa_512 [part] at (1150, 250, 200) mm
  - Placa_513 [part] at (1150, 250, 200) mm
  - Placa_514 [part] at (1150, 250, 200) mm
  - Placa_515 [part] at (1150, 250, 200) mm
  - Disco_516 [part] at (1250, 230, 200) mm
  - Placa_517 [part] at (1150, 250, 200) mm
  - Placa_518 [part] at (1150, 250, 200) mm
  - Placa_519 [part] at (1150, 250, 200) mm
  - Disco_520 [part] at (1250, 230, 200) mm
  - Placa_521 [part] at (1150, 250, 200) mm
  - Placa_522 [part] at (1150, 250, 200) mm
  - Disco_523 [part] at (1250, 230, 200) mm
  - Placa_524 [part] at (1150, 250, 200) mm
  - Disco_525 [part] at (1250, 230, 200) mm
  - Placa_526 [part] at (1150, 250, 200) mm
  - Placa_527 [part] at (1150, 250, 200) mm
  - Placa_528 [part] at (1150, 250, 200) mm
  - Placa_529 [part] at (1150, 250, 200) mm
  - Disco_530 [part] at (1250, 230, 200) mm
  - Disco_531 [part] at (1250, 230, 200) mm
  - Disco_532 [part] at (1250, 230, 200) mm
  - Disco_533 [part] at (1250, 230, 200) mm
  - Disco_534 [part] at (1250, 230, 200) mm
  - Disco_535 [part] at (1250, 230, 200) mm
  - Disco_536 [part] at (1250, 230, 200) mm
  - Placa_537 [part] at (1150, 250, 200) mm
  - Placa_538 [part] at (1150, 250, 200) mm
  - Disco_539 [part] at (1250, 230, 200) mm
  - Placa_540 [part] at (1150, 250, 200) mm
  - Disco_541 [part] at (1250, 230, 200) mm
  - Disco_542 [part] at (1250, 230, 200) mm
  - Placa_543 [part] at (1150, 250, 200) mm
  - Disco_544 [part] at (1250, 230, 200) mm
  - Disco_545 [part] at (1250, 230, 200) mm
  - Placa_546 [part] at (1150, 250, 200) mm
  - Disco_547 [part] at (1250, 230, 200) mm
  - Disco_548 [part] at (1250, 230, 200) mm
  - Disco_549 [part] at (1250, 230, 200) mm
  - Placa_550 [part] at (1150, 250, 200) mm
  - Placa_551 [part] at (1150, 250, 200) mm
  - Placa_552 [part] at (1150, 250, 200) mm
  - Placa_553 [part] at (1150, 250, 200) mm
  - Disco_554 [part] at (1250, 230, 200) mm
  - Disco_555 [part] at (1250, 230, 200) mm
  - Placa_556 [part] at (1150, 250, 200) mm
  - Disco_557 [part] at (1250, 230, 200) mm
  - Disco_558 [part] at (1250, 230, 200) mm
  - Disco_559 [part] at (1250, 230, 200) mm
  - Placa_560 [part] at (1150, 250, 200) mm
  - Disco_561 [part] at (1250, 230, 200) mm
  - Placa_562 [part] at (1150, 250, 200) mm
  - Placa_563 [part] at (1150, 250, 200) mm
  - Placa_564 [part] at (1150, 250, 200) mm
  - Placa_565 [part] at (1150, 250, 200) mm
  - Placa_566 [part] at (1150, 250, 200) mm
  - Placa_567 [part] at (1150, 250, 200) mm
  - Disco_568 [part] at (1250, 230, 200) mm
  - Disco_569 [part] at (1250, 230, 200) mm
  - Placa_570 [part] at (1150, 250, 200) mm
  - Disco_571 [part] at (1250, 230, 200) mm
  - Disco_572 [part] at (1250, 230, 200) mm
  - Placa_573 [part] at (1150, 250, 200) mm
  - Placa_574 [part] at (1150, 250, 200) mm
  - Disco_575 [part] at (1250, 230, 200) mm
  - Placa_576 [part] at (1150, 250, 200) mm
  - Placa_577 [part] at (1150, 250, 200) mm
  - Placa_578 [part] at (1150, 250, 200) mm
  - Disco_579 [part] at (1250, 230, 200) mm
  - Placa_580 [part] at (1150, 250, 200) mm
  - Disco_581 [part] at (1250, 230, 200) mm
  - Placa_582 [part] at (1150, 250, 200) mm
  - Placa_583 [part] at (1150, 250, 200) mm
  - Disco_584 [part] at (1250, 230, 200) mm
  - Disco_585 [part] at (1250, 230, 200) mm
  - Placa_586 [part] at (1150, 250, 200) mm
  - Disco_587 [part] at (1250, 230, 200) mm
  - Placa_588 [part] at (1150, 250, 200) mm
  - Disco_589 [part] at (1250, 230, 200) mm
  - Placa_590 [part] at (1150, 250, 200) mm
  - Placa_591 [part] at (1150, 250, 200) mm
  - Placa_592 [part] at (1150, 250, 200) mm
  - Placa_593 [part] at (1150, 250, 200) mm
  - Disco_594 [part] at (1250, 230, 200) mm
  - Placa_595 [part] at (1150, 250, 200) mm
  - Disco_596 [part] at (1250, 230, 200) mm
  - Placa_597 [part] at (1150, 250, 200) mm
  - Placa_598 [part] at (1150, 250, 200) mm
  - Disco_600 [part] at (1250, 230, 200) mm
  - Placa_601 [part] at (1150, 250, 200) mm
  - Placa_602 [part] at (1150, 250, 200) mm
  - Placa_603 [part] at (1150, 250, 200) mm
  - Disco_604 [part] at (1250, 230, 200) mm
  - Disco_605 [part] at (1250, 230, 200) mm
  - Placa_606 [part] at (1150, 250, 200) mm
  - Placa_607 [part] at (1150, 250, 200) mm
  - Disco_608 [part] at (1250, 230, 200) mm
  - Disco_609 [part] at (1250, 230, 200) mm
  - Disco_610 [part] at (1250, 230, 200) mm
  - Placa_611 [part] at (1150, 250, 200) mm
  - Disco_612 [part] at (1250, 230, 200) mm
  - Placa_613 [part] at (1150, 250, 200) mm
  - Disco_614 [part] at (1250, 230, 200) mm
  - Placa_615 [part] at (1150, 250, 200) mm
  - Disco_616 [part] at (1250, 230, 200) mm
  - Disco_617 [part] at (1250, 230, 200) mm
  - Disco_618 [part] at (1250, 230, 200) mm
  - Disco_619 [part] at (1250, 230, 200) mm
  - Disco_620 [part] at (1250, 230, 200) mm
  - Placa_621 [part] at (1150, 250, 200) mm
  - Placa_622 [part] at (1150, 250, 200) mm
  - Placa_624 [part] at (1150, 250, 200) mm
  - Placa_625 [part] at (1150, 250, 200) mm
  - Placa_626 [part] at (1150, 250, 200) mm
  - Placa_627 [part] at (1150, 250, 200) mm
  - Disco_628 [part] at (1250, 230, 200) mm
  - Disco_629 [part] at (1250, 230, 200) mm
  - Placa_630 [part] at (1150, 250, 200) mm
  - Disco_631 [part] at (1250, 230, 200) mm
  - Placa_632 [part] at (1150, 250, 200) mm
  - Placa_633 [part] at (1150, 250, 200) mm
  - Placa_634 [part] at (1150, 250, 200) mm
  - Disco_635 [part] at (1250, 230, 200) mm
  - Disco_636 [part] at (1250, 230, 200) mm
  - Disco_637 [part] at (1250, 230, 200) mm
  - Disco_638 [part] at (1250, 230, 200) mm
  - Placa_639 [part] at (1150, 250, 200) mm
  - Placa_640 [part] at (1150, 250, 200) mm
  - Placa_641 [part] at (1150, 250, 200) mm
  - Disco_642 [part] at (1250, 230, 200) mm
  - Placa_643 [part] at (1150, 250, 200) mm
  - Placa_644 [part] at (1150, 250, 200) mm
  - Disco_645 [part] at (1250, 230, 200) mm
  - Disco_646 [part] at (1250, 230, 200) mm
  - Disco_648 [part] at (1250, 230, 200) mm
  - Placa_649 [part] at (1150, 250, 200) mm
  - Placa_650 [part] at (1150, 250, 200) mm
  - Placa_651 [part] at (1150, 250, 200) mm
  - Disco_652 [part] at (1250, 230, 200) mm
  - Placa_653 [part] at (1150, 250, 200) mm
  - Disco_654 [part] at (1250, 230, 200) mm
  - Placa_655 [part] at (1150, 250, 200) mm
  - Placa_656 [part] at (1150, 250, 200) mm
  - Disco_657 [part] at (1250, 230, 200) mm
  - Placa_658 [part] at (1150, 250, 200) mm
  - Placa_659 [part] at (1150, 250, 200) mm
  - Placa_660 [part] at (1150, 250, 200) mm
  - Disco_661 [part] at (1250, 230, 200) mm
  - Placa_662 [part] at (1150, 250, 200) mm
  - Disco_663 [part] at (1250, 230, 200) mm
  - Disco_664 [part] at (1250, 230, 200) mm
  - Disco_665 [part] at (1250, 230, 200) mm
  - Placa_666 [part] at (1150, 250, 200) mm
  - Placa_667 [part] at (1150, 250, 200) mm
  - Placa_668 [part] at (1150, 250, 200) mm
  - Placa_669 [part] at (1150, 250, 200) mm
  - Disco_670 [part] at (1250, 230, 200) mm
  - Disco_672 [part] at (1250, 230, 200) mm
  - Placa_673 [part] at (1150, 250, 200) mm
  - Placa_674 [part] at (1150, 250, 200) mm
  - Disco_675 [part] at (1250, 230, 200) mm
  - Placa_676 [part] at (1150, 250, 200) mm
  - Disco_677 [part] at (1250, 230, 200) mm
  - Placa_678 [part] at (1150, 250, 200) mm
  - Disco_679 [part] at (1250, 230, 200) mm
  - Placa_680 [part] at (1150, 250, 200) mm
  - Placa_681 [part] at (1150, 250, 200) mm
  - Disco_682 [part] at (1250, 230, 200) mm
  - Placa_683 [part] at (1150, 250, 200) mm
  - Disco_684 [part] at (1250, 230, 200) mm
  - Placa_685 [part] at (1150, 250, 200) mm
  - Disco_686 [part] at (1250, 230, 200) mm
  - Disco_687 [part] at (1250, 230, 200) mm
  - Disco_688 [part] at (1250, 230, 200) mm
  - Disco_689 [part] at (1250, 230, 200) mm
  - Disco_690 [part] at (1250, 230, 200) mm
  - Placa_691 [part] at (1150, 250, 200) mm
  - Placa_692 [part] at (1150, 250, 200) mm
  - Disco_693 [part] at (1250, 230, 200) mm
  - Disco_694 [part] at (1250, 230, 200) mm
  - Placa_695 [part] at (1150, 250, 200) mm
  - Disco_696 [part] at (1250, 230, 200) mm
  - Disco_707 [part] at (1250, 230, 200) mm
  - Placa_708 [part] at (1150, 250, 200) mm
  - Placa_709 [part] at (1150, 250, 200) mm
  - Disco_710 [part] at (1250, 230, 200) mm
  - Placa_711 [part] at (1150, 250, 200) mm
  - Placa_712 [part] at (1150, 250, 200) mm
  - Disco_713 [part] at (1250, 230, 200) mm
  - Disco_714 [part] at (1250, 230, 200) mm
  - Placa_715 [part] at (1150, 250, 200) mm
  - Disco_716 [part] at (1250, 230, 200) mm
  - Placa_717 [part] at (1150, 250, 200) mm
  - Placa_718 [part] at (1150, 250, 200) mm
  - Placa_720 [part] at (1150, 250, 200) mm
  - Disco_721 [part] at (1250, 230, 200) mm
  - Disco_722 [part] at (1250, 230, 200) mm
  - Placa_723 [part] at (1150, 250, 200) mm
  - Disco_724 [part] at (1250, 230, 200) mm
  - Disco_725 [part] at (1250, 230, 200) mm
  - Disco_726 [part] at (1250, 230, 200) mm
  - Placa_727 [part] at (1150, 250, 200) mm
  - Placa_728 [part] at (1150, 250, 200) mm
  - Disco_729 [part] at (1250, 230, 200) mm
  - Disco_730 [part] at (1250, 230, 200) mm
  - Disco_731 [part] at (1250, 230, 200) mm
  - Placa_732 [part] at (1150, 250, 200) mm
  - Disco_733 [part] at (1250, 230, 200) mm
  - Disco_734 [part] at (1250, 230, 200) mm
  - Disco_735 [part] at (1250, 230, 200) mm
  - Placa_736 [part] at (1150, 250, 200) mm
  - Disco_737 [part] at (1250, 230, 200) mm
  - Disco_738 [part] at (1250, 230, 200) mm
  - Placa_739 [part] at (1150, 250, 200) mm
  - Placa_740 [part] at (1150, 250, 200) mm
  - Placa_741 [part] at (1150, 250, 200) mm
  - Disco_742 [part] at (1250, 230, 200) mm
  - Placa_743 [part] at (1146.4, 250, 200) mm
  - Disco_744 [part] at (1250, 230, 200) mm
  - Placa_745 [part] at (1150, 250, 200) mm
  - Disco_746 [part] at (1250, 230, 200) mm
  - Disco_747 [part] at (1250, 230, 200) mm
  - Disco_748 [part] at (1250, 230, 200) mm
  - Disco_749 [part] at (1250, 230, 200) mm
  - Disco_750 [part] at (1250, 230, 200) mm
  - Disco_751 [part] at (1250, 230, 200) mm
  - Placa_752 [part] at (1150, 250, 200) mm
  - Placa_753 [part] at (1150, 250, 200) mm
  - Placa_754 [part] at (1150, 250, 200) mm
  - Placa_755 [part] at (1150, 250, 200) mm
  - Disco_756 [part] at (1250, 230, 200) mm
  - Disco_757 [part] at (1250, 230, 200) mm
  - Disco_758 [part] at (1250, 230, 200) mm
  - Disco_759 [part] at (1250, 230, 200) mm
  - Placa_760 [part] at (1150, 250, 200) mm
  - Placa_761 [part] at (1150, 250, 200) mm
  - Placa_762 [part] at (1150, 250, 200) mm
  - Placa_763 [part] at (1150, 250, 200) mm
  - Placa_764 [part] at (1150, 250, 200) mm
  - Placa_765 [part] at (1150, 250, 200) mm
  - Disco_766 [part] at (1250, 230, 200) mm
  - Placa_767 [part] at (1146.4, 250, 200) mm
  - Disco_768 [part] at (1250, 230, 200) mm
  - Disco_769 [part] at (1250, 230, 200) mm
  - Placa_770 [part] at (1150, 250, 200) mm
  - Placa_771 [part] at (1150, 250, 200) mm
  - Placa_772 [part] at (1150, 250, 200) mm
  - Placa_773 [part] at (1150, 250, 200) mm
  - Placa_774 [part] at (1150, 250, 200) mm
  - Disco_775 [part] at (1250, 230, 200) mm
  - Placa_776 [part] at (1150, 250, 200) mm
  - Placa_777 [part] at (1150, 250, 200) mm
  - Placa_778 [part] at (1150, 250, 200) mm
  - Placa_779 [part] at (1150, 250, 200) mm
  - Disco_780 [part] at (1250, 230, 200) mm
  - Disco_781 [part] at (1250, 230, 200) mm
  - Disco_782 [part] at (1250, 230, 200) mm
  - Disco_783 [part] at (1250, 230, 200) mm
  - Placa_784 [part] at (1150, 250, 200) mm
  - Placa_785 [part] at (1150, 250, 200) mm
  - Placa_786 [part] at (1150, 250, 200) mm
  - Placa_787 [part] at (1150, 250, 200) mm
  - Disco_788 [part] at (1250, 230, 200) mm
  - Disco_789 [part] at (1250, 230, 200) mm
  - Placa_790 [part] at (1150, 250, 200) mm
  - Placa_791 [part] at (1150, 250, 200) mm
  - Disco_792 [part] at (1250, 230, 200) mm
  - Disco_793 [part] at (1250, 230, 200) mm
  - Placa_794 [part] at (1150, 250, 200) mm
  - Disco_795 [part] at (1250, 230, 200) mm
  - Disco_796 [part] at (1250, 230, 200) mm
  - Placa_797 [part] at (1150, 250, 200) mm
  - Disco_798 [part] at (1250, 230, 200) mm
  - Disco_799 [part] at (1250, 230, 200) mm
  - Disco_800 [part] at (1250, 230, 200) mm
  - Placa_801 [part] at (1150, 250, 200) mm
  - Placa_802 [part] at (1150, 250, 200) mm
  - Disco_803 [part] at (1250, 230, 200) mm
  - Disco_804 [part] at (1250, 230, 200) mm
  - Placa_805 [part] at (1150, 250, 200) mm
  - Placa_806 [part] at (1150, 250, 200) mm
  - Placa_807 [part] at (1150, 250, 200) mm
  - Placa_808 [part] at (1150, 250, 200) mm
  - Placa_809 [part] at (1150, 250, 200) mm
  - Disco_810 [part] at (1250, 230, 200) mm
  - Placa_811 [part] at (1150, 250, 200) mm
  - Disco_812 [part] at (1250, 230, 200) mm
  - Disco_813 [part] at (1250, 230, 200) mm
  - Placa_814 [part] at (1150, 250, 200) mm
  - Placa_815 [part] at (1150, 250, 200) mm
  - Disco_816 [part] at (1250, 230, 200) mm
  - Disco_817 [part] at (1250, 230, 200) mm
  - Placa_818 [part] at (1150, 250, 200) mm
  - Placa_819 [part] at (1150, 250, 200) mm
  - Placa_820 [part] at (1150, 250, 200) mm
  - Disco_821 [part] at (1250, 230, 200) mm
  - Disco_822 [part] at (1250, 230, 200) mm
  - Disco_823 [part] at (1250, 230, 200) mm
  - Disco_824 [part] at (1250, 230, 200) mm
  - Placa_825 [part] at (1150, 250, 200) mm
  - Disco_826 [part] at (1250, 230, 200) mm
  - Disco_827 [part] at (1250, 230, 200) mm
  - Disco_828 [part] at (1250, 230, 200) mm
  - Placa_829 [part] at (1150, 250, 200) mm
  - Placa_830 [part] at (1150, 250, 200) mm
  - Disco_831 [part] at (1250, 230, 200) mm
  - Placa_832 [part] at (1150, 250, 200) mm
  - Disco_833 [part] at (1250, 230, 200) mm
  - Disco_834 [part] at (1250, 230, 200) mm
  - Placa_835 [part] at (1150, 250, 200) mm
  - Disco_836 [part] at (1250, 230, 200) mm
  - Disco_837 [part] at (1250, 230, 200) mm
  - Placa_838 [part] at (1150, 250, 200) mm
  - Placa_839 [part] at (1150, 250, 200) mm
  - Disco_840 [part] at (1250, 230, 200) mm
  - Disco_841 [part] at (1250, 230, 200) mm
  - Disco_842 [part] at (1250, 230, 200) mm
  - Placa_843 [part] at (1150, 250, 200) mm
  - Disco_844 [part] at (1250, 230, 200) mm
  - Disco_845 [part] at (1250, 230, 200) mm
  - Placa_846 [part] at (1150, 250, 200) mm
  - Disco_847 [part] at (1250, 230, 200) mm
  - Disco_848 [part] at (1250, 230, 200) mm
  - Disco_849 [part] at (1250, 230, 200) mm
  - Placa_850 [part] at (1150, 250, 200) mm
  - Placa_851 [part] at (1150, 250, 200) mm
  - Placa_852 [part] at (1150, 250, 200) mm
  - Disco_853 [part] at (1250, 230, 200) mm
  - Placa_854 [part] at (1150, 250, 200) mm
  - Disco_855 [part] at (1250, 230, 200) mm
  - Disco_856 [part] at (1250, 230, 200) mm
  - Disco_857 [part] at (1250, 230, 200) mm
  - Placa_858 [part] at (1150, 250, 200) mm
  - Placa_859 [part] at (1150, 250, 200) mm
  - Placa_860 [part] at (1150, 250, 200) mm
  - Disco_861 [part] at (1250, 230, 200) mm
  - Placa_862 [part] at (1150, 250, 200) mm
  - Disco_863 [part] at (1250, 230, 200) mm
  - Placa_864 [part] at (1150, 250, 200) mm
  - Placa_865 [part] at (1150, 250, 200) mm
  - Placa_866 [part] at (1150, 250, 200) mm
  - Placa_867 [part] at (1150, 250, 200) mm
  - Placa_868 [part] at (1150, 250, 200) mm
  - Disco_869 [part] at (1250, 230, 200) mm
  - Disco_870 [part] at (1250, 230, 200) mm
  - Disco_871 [part] at (1250, 230, 200) mm
  - Placa_872 [part] at (1150, 250, 200) mm
  - Placa_873 [part] at (1150, 250, 200) mm
  - Disco_874 [part] at (1250, 230, 200) mm
  - Disco_875 [part] at (1250, 230, 200) mm
  - Disco_876 [part] at (1250, 230, 200) mm
  - Placa_877 [part] at (1150, 250, 200) mm
  - Disco_878 [part] at (1250, 230, 200) mm
  - Placa_879 [part] at (1150, 250, 200) mm
  - Disco_880 [part] at (1250, 230, 200) mm
  - Disco_881 [part] at (1250, 230, 200) mm
  - Placa_882 [part] at (1150, 250, 200) mm
  - Placa_883 [part] at (1150, 250, 200) mm
  - Placa_884 [part] at (1150, 250, 200) mm
  - Disco_885 [part] at (1250, 230, 200) mm
  - Disco_886 [part] at (1250, 230, 200) mm
  - Disco_887 [part] at (1250, 230, 200) mm
  - Placa_888 [part] at (1150, 250, 200) mm
  - Disco_889 [part] at (1250, 230, 200) mm
  - Disco_890 [part] at (1250, 230, 200) mm
  - Placa_891 [part] at (1150, 250, 200) mm
  - Disco_892 [part] at (1250, 230, 200) mm
  - Disco_893 [part] at (1250, 230, 200) mm
  - Disco_894 [part] at (1250, 230, 200) mm
  - Placa_895 [part] at (1150, 250, 200) mm
  - Placa_896 [part] at (1150, 250, 200) mm
  - Placa_897 [part] at (1150, 250, 200) mm
  - Placa_898 [part] at (1150, 250, 200) mm
  - Disco_899 [part] at (1250, 230, 200) mm
  - Disco_900 [part] at (1250, 230, 200) mm
  - Disco_901 [part] at (1250, 230, 200) mm
  - Disco_902 [part] at (1250, 230, 200) mm
  - Disco_903 [part] at (1250, 230, 200) mm
  - Disco_904 [part] at (1250, 230, 200) mm
  - Placa_905 [part] at (1150, 250, 200) mm
  - Disco_906 [part] at (1250, 230, 200) mm
  - Disco_907 [part] at (1250, 230, 200) mm
  - Placa_908 [part] at (1150, 250, 200) mm
  - Disco_909 [part] at (1246.4, 230, 200) mm
  - Disco_910 [part] at (1250, 230, 200) mm
  - Placa_911 [part] at (1150, 250, 200) mm
  - Disco_912 [part] at (1250, 230, 200) mm
  - Placa_913 [part] at (1150, 250, 200) mm
  - Placa_914 [part] at (1150, 250, 200) mm
  - Disco_915 [part] at (1250, 230, 200) mm
  - Placa_916 [part] at (1150, 250, 200) mm
  - Placa_917 [part] at (1150, 250, 200) mm
  - Disco_918 [part] at (1250, 230, 200) mm
  - Placa_919 [part] at (1150, 250, 200) mm
  - Placa_920 [part] at (1150, 250, 200) mm
  - Placa_921 [part] at (1150, 250, 200) mm
  - Placa_922 [part] at (1150, 250, 200) mm
  - Placa_923 [part] at (1150, 250, 200) mm
  - Placa_924 [part] at (1150, 250, 200) mm
  - Disco_925 [part] at (1250, 230, 200) mm
  - Placa_926 [part] at (1150, 250, 200) mm
  - Disco_927 [part] at (1250, 230, 200) mm
  - Placa_928 [part] at (1150, 250, 200) mm
  - Placa_929 [part] at (1150, 250, 200) mm
  - Placa_930 [part] at (1150, 250, 200) mm
  - Disco_931 [part] at (1250, 230, 200) mm
  - Placa_932 [part] at (1150, 250, 200) mm
  - Placa_933 [part] at (1146.4, 250, 200) mm
  - Placa_934 [part] at (1150, 250, 200) mm
  - Placa_935 [part] at (1150, 250, 200) mm
  - Placa_936 [part] at (1150, 250, 200) mm
  - Placa_937 [part] at (1150, 250, 200) mm
  - Placa_938 [part] at (1150, 250, 200) mm
  - Disco_939 [part] at (1250, 230, 200) mm
  - Placa_940 [part] at (1150, 250, 200) mm
  - Disco_941 [part] at (1250, 230, 200) mm
  - Disco_942 [part] at (1250, 230, 200) mm
  - Placa_943 [part] at (1150, 250, 200) mm
  - Placa_944 [part] at (1150, 250, 200) mm
  - Placa_945 [part] at (1150, 250, 200) mm
  - Placa_946 [part] at (1150, 250, 200) mm
  - Disco_947 [part] at (1250, 230, 200) mm
  - Placa_948 [part] at (1150, 250, 200) mm
  - Disco_949 [part] at (1250, 230, 200) mm
  - Disco_950 [part] at (1250, 230, 200) mm
  - Placa_951 [part] at (1150, 250, 200) mm
  - Placa_952 [part] at (1150, 250, 200) mm
  - Disco_953 [part] at (1250, 230, 200) mm
  - Disco_954 [part] at (1250, 230, 200) mm
  - Placa_955 [part] at (1150, 250, 200) mm
  - Disco_956 [part] at (1250, 230, 200) mm
  - Disco_957 [part] at (1246.4, 230, 200) mm
  - Disco_958 [part] at (1250, 230, 200) mm
  - Placa_959 [part] at (1150, 250, 200) mm
  - Placa_960 [part] at (1150, 250, 200) mm
  - Placa_961 [part] at (1150, 250, 200) mm
  - Placa_962 [part] at (1150, 250, 200) mm
  - Disco_963 [part] at (1250, 230, 200) mm
  - Disco_964 [part] at (1250, 230, 200) mm
  - Placa_965 [part] at (1150, 250, 200) mm
  - Placa_966 [part] at (1150, 250, 200) mm
  - Disco_967 [part] at (1250, 230, 200) mm
  - Disco_968 [part] at (1250, 230, 200) mm
  - Placa_969 [part] at (1150, 250, 200) mm
  - Placa_970 [part] at (1150, 250, 200) mm
  - Placa_971 [part] at (1150, 250, 200) mm
  - Disco_972 [part] at (1250, 230, 200) mm
  - Disco_973 [part] at (1250, 230, 200) mm
  - Placa_974 [part] at (1150, 250, 200) mm
  - Placa_975 [part] at (1150, 250, 200) mm
  - Disco_976 [part] at (1250, 230, 200) mm
  - Disco_977 [part] at (1250, 230, 200) mm
  - Placa_978 [part] at (1150, 250, 200) mm
  - Placa_979 [part] at (1150, 250, 200) mm
  - Placa_980 [part] at (1150, 250, 200) mm
  - Disco_981 [part] at (1246.4, 230, 200) mm
  - Placa_982 [part] at (1150, 250, 200) mm
  - Disco_983 [part] at (1250, 230, 200) mm
  - Placa_984 [part] at (1150, 250, 200) mm
  - Placa_985 [part] at (1150, 250, 200) mm
  - Placa_986 [part] at (1150, 250, 200) mm
  - Disco_987 [part] at (1250, 230, 200) mm
  - Placa_988 [part] at (1150, 250, 200) mm
  - Disco_989 [part] at (1250, 230, 200) mm
  - Placa_990 [part] at (1150, 250, 200) mm
  - Disco_991 [part] at (1250, 230, 200) mm
  - Placa_992 [part] at (1150, 250, 200) mm
  - Disco_993 [part] at (1250, 230, 200) mm
  - Disco_994 [part] at (1250, 230, 200) mm
  - Placa_995 [part] at (1150, 250, 200) mm
  - Placa_996 [part] at (1150, 250, 200) mm
  - Disco_997 [part] at (1250, 230, 200) mm
  - Disco_998 [part] at (1250, 230, 200) mm
  - Placa_999 [part] at (1150, 250, 200) mm
  - Disco_1000 [part] at (1250, 230, 200) mm
  - Disco_1001 [part] at (1250, 230, 200) mm
  - Disco_1002 [part] at (1250, 230, 200) mm
  - Placa_1003 [part] at (1150, 250, 200) mm
  - Disco_1004 [part] at (1250, 230, 200) mm
  - Disco_1005 [part] at (1246.4, 230, 200) mm
  - Disco_1006 [part] at (1250, 230, 200) mm
  - Placa_1007 [part] at (1150, 250, 200) mm
  - Placa_1008 [part] at (1150, 250, 200) mm
  - Placa_1009 [part] at (1150, 250, 200) mm
  - Disco_1010 [part] at (1250, 230, 200) mm
  - Disco_1011 [part] at (1250, 230, 200) mm
  - Placa_1012 [part] at (1150, 250, 200) mm
  - Disco_1013 [part] at (1250, 230, 200) mm
  - Placa_1014 [part] at (1150, 250, 200) mm
  - Placa_1015 [part] at (1150, 250, 200) mm
  - Disco_1016 [part] at (1250, 230, 200) mm
  - Disco_1017 [part] at (1250, 230, 200) mm
  - Placa_1018 [part] at (1150, 250, 200) mm
  - Placa_1019 [part] at (1150, 250, 200) mm
  - Disco_1020 [part] at (1250, 230, 200) mm
  - Placa_1021 [part] at (1150, 250, 200) mm
  - Placa_1022 [part] at (1150, 250, 200) mm
  - Disco_1023 [part] at (1250, 230, 200) mm
  - Placa_1024 [part] at (1150, 250, 200) mm
  - Disco_1025 [part] at (1250, 230, 200) mm
  - Disco_1026 [part] at (1250, 230, 200) mm
  - Disco_1027 [part] at (1250, 230, 200) mm
  - Placa_1028 [part] at (1150, 250, 200) mm
  - Placa_1029 [part] at (1146.4, 250, 200) mm
  - Placa_1030 [part] at (1150, 250, 200) mm
  - Disco_1031 [part] at (1250, 230, 200) mm
  - Disco_1032 [part] at (1250, 230, 200) mm
  - Placa_1033 [part] at (1150, 250, 200) mm
  - Placa_1034 [part] at (1150, 250, 200) mm
  - Placa_1035 [part] at (1150, 250, 200) mm
  - Disco_1036 [part] at (1250, 230, 200) mm
  - Placa_1037 [part] at (1150, 250, 200) mm
  - Disco_1038 [part] at (1250, 230, 200) mm
  - Disco_1039 [part] at (1250, 230, 200) mm
  - Disco_1040 [part] at (1250, 230, 200) mm
  - Disco_1041 [part] at (1250, 230, 200) mm
  - Placa_1042 [part] at (1150, 250, 200) mm
  - Placa_1043 [part] at (1150, 250, 200) mm
  - Placa_1044 [part] at (1150, 250, 200) mm
  - Placa_1045 [part] at (1150, 250, 200) mm
  - Placa_1046 [part] at (1150, 250, 200) mm
  - Disco_1047 [part] at (1250, 230, 200) mm
  - Disco_1048 [part] at (1250, 230, 200) mm
  - Placa_1049 [part] at (1150, 250, 200) mm
  - Placa_1050 [part] at (1150, 250, 200) mm
  - Placa_1051 [part] at (1150, 250, 200) mm
  - Disco_1052 [part] at (1250, 230, 200) mm
  - Placa_1053 [part] at (1146.4, 250, 200) mm
  - Placa_1054 [part] at (1150, 250, 200) mm
  - Disco_1055 [part] at (1250, 230, 200) mm
  - Disco_1056 [part] at (1250, 230, 200) mm
  - Placa_1057 [part] at (1150, 250, 200) mm
  - Disco_1058 [part] at (1250, 230, 200) mm
  - Disco_1059 [part] at (1250, 230, 200) mm
  - Disco_1060 [part] at (1250, 230, 200) mm
  - Disco_1061 [part] at (1250, 230, 200) mm
  - Placa_1062 [part] at (1150, 250, 200) mm
  - Placa_1063 [part] at (1150, 250, 200) mm
  - Placa_1064 [part] at (1150, 250, 200) mm
  - Placa_1065 [part] at (1150, 250, 200) mm
  - Placa_1066 [part] at (1150, 250, 200) mm
  - Placa_1067 [part] at (1150, 250, 200) mm
  - Disco_1068 [part] at (1250, 230, 200) mm
  - Placa_1069 [part] at (1150, 250, 200) mm
  - Disco_1070 [part] at (1250, 230, 200) mm
  - Disco_1071 [part] at (1250, 230, 200) mm
  - Placa_1072 [part] at (1150, 250, 200) mm
  - Placa_1073 [part] at (1150, 250, 200) mm
  - Disco_1074 [part] at (1250, 230, 200) mm
  - Disco_1075 [part] at (1250, 230, 200) mm
  - Disco_1076 [part] at (1250, 230, 200) mm
  - Disco_1077 [part] at (1246.4, 230, 200) mm
  - Disco_1078 [part] at (1250, 230, 200) mm
  - Disco_1079 [part] at (1250, 230, 200) mm
  - Disco_1080 [part] at (1250, 230, 200) mm
  - Disco_1081 [part] at (1250, 230, 200) mm
  - Placa_1082 [part] at (1150, 250, 200) mm
  - Placa_1083 [part] at (1150, 250, 200) mm
  - Placa_1084 [part] at (1150, 250, 200) mm
  - Disco_1085 [part] at (1250, 230, 200) mm
  - Disco_1086 [part] at (1250, 230, 200) mm
  - Disco_1087 [part] at (1250, 230, 200) mm
  - Disco_1088 [part] at (1250, 230, 200) mm
  - Placa_1089 [part] at (1150, 250, 200) mm
  - Disco_1090 [part] at (1250, 230, 200) mm
  - Placa_1091 [part] at (1150, 250, 200) mm
  - Placa_1092 [part] at (1150, 250, 200) mm
  - Placa_1093 [part] at (1150, 250, 200) mm
  - Placa_1094 [part] at (1150, 250, 200) mm
  - Disco_1095 [part] at (1250, 230, 200) mm
  - Disco_1096 [part] at (1250, 230, 200) mm
  - Placa_1097 [part] at (1150, 250, 200) mm
  - Placa_1098 [part] at (1150, 250, 200) mm
  - Disco_1099 [part] at (1250, 230, 200) mm
  - Placa_1100 [part] at (1150, 250, 200) mm
  - Disco_1101 [part] at (1246.4, 230, 200) mm
  - Placa_1102 [part] at (1150, 250, 200) mm
  - Placa_1103 [part] at (1150, 250, 200) mm
  - Placa_1104 [part] at (1150, 250, 200) mm
  - Placa_1105 [part] at (1150, 250, 200) mm
  - Placa_1106 [part] at (1150, 250, 200) mm
  - Placa_1107 [part] at (1150, 250, 200) mm
  - Placa_1108 [part] at (1150, 250, 200) mm
  - Placa_1109 [part] at (1150, 250, 200) mm
  - Disco_1110 [part] at (1250, 230, 200) mm
  - Disco_1111 [part] at (1250, 230, 200) mm
  - Disco_1112 [part] at (1250, 230, 200) mm
  - Placa_1113 [part] at (1150, 250, 200) mm
  - Placa_1114 [part] at (1150, 250, 200) mm
  - Disco_1115 [part] at (1250, 230, 200) mm
  - Disco_1116 [part] at (1250, 230, 200) mm
  - Placa_1117 [part] at (1150, 250, 200) mm
  - Disco_1118 [part] at (1250, 230, 200) mm
  - Placa_1119 [part] at (1150, 250, 200) mm
  - Placa_1120 [part] at (1150, 250, 200) mm
  - Placa_1121 [part] at (1150, 250, 200) mm
  - Disco_1122 [part] at (1250, 230, 200) mm
  - Placa_1123 [part] at (1150, 250, 200) mm
  - Disco_1124 [part] at (1250, 230, 200) mm
  - Disco_1125 [part] at (1246.4, 230, 200) mm
  - Disco_1126 [part] at (1250, 230, 200) mm
  - Disco_1127 [part] at (1250, 230, 200) mm
  - Placa_1128 [part] at (1150, 250, 200) mm
  - Placa_1129 [part] at (1150, 250, 200) mm
  - Placa_1130 [part] at (1150, 250, 200) mm
  - Disco_1131 [part] at (1250, 230, 200) mm
  - Disco_1132 [part] at (1250, 230, 200) mm
  - Disco_1133 [part] at (1250, 230, 200) mm
  - Disco_1134 [part] at (1250, 230, 200) mm
  - Disco_1135 [part] at (1250, 230, 200) mm
  - Disco_1136 [part] at (1250, 230, 200) mm
  - Disco_1137 [part] at (1250, 230, 200) mm
  - Disco_1138 [part] at (1250, 230, 200) mm
  - Disco_1139 [part] at (1250, 230, 200) mm
  - Placa_1140 [part] at (1150, 250, 200) mm
  - Disco_1141 [part] at (1250, 230, 200) mm
  - Placa_1142 [part] at (1150, 250, 200) mm
  - Placa_1143 [part] at (1150, 250, 200) mm
  - Disco_1144 [part] at (1250, 230, 200) mm
  - Disco_1145 [part] at (1250, 230, 200) mm
  - Disco_1146 [part] at (1250, 230, 200) mm
  - Placa_1147 [part] at (1150, 250, 200) mm
  - Placa_1148 [part] at (1150, 250, 200) mm
  - Placa_1149 [part] at (1146.4, 250, 200) mm
  - Placa_1150 [part] at (1150, 250, 200) mm
  - Disco_1151 [part] at (1250, 230, 200) mm
  - Disco_1152 [part] at (1250, 230, 200) mm
  - Disco_1153 [part] at (1250, 230, 200) mm
  - Placa_1154 [part] at (1150, 250, 200) mm
  - Disco_1155 [part] at (1250, 230, 200) mm
  - Placa_1156 [part] at (1150, 250, 200) mm
  - Disco_1157 [part] at (1250, 230, 200) mm
  - Disco_1158 [part] at (1250, 230, 200) mm
  - Disco_1159 [part] at (1250, 230, 200) mm
  - Disco_1160 [part] at (1250, 230, 200) mm
  - Disco_1161 [part] at (1250, 230, 200) mm
  - Disco_1162 [part] at (1250, 230, 200) mm
  - Placa_1163 [part] at (1150, 250, 200) mm
  - Placa_1164 [part] at (1150, 250, 200) mm
  - Placa_1165 [part] at (1150, 250, 200) mm
  - Placa_1166 [part] at (1150, 250, 200) mm
  - Disco_1167 [part] at (1250, 230, 200) mm
  - Placa_1168 [part] at (1150, 250, 200) mm
  - Placa_1169 [part] at (1150, 250, 200) mm
  - Placa_1170 [part] at (1150, 250, 200) mm
  - Disco_1171 [part] at (1250, 230, 200) mm
  - Placa_1172 [part] at (1150, 250, 200) mm
  - Disco_1173 [part] at (1246.4, 230, 200) mm
  - Placa_1174 [part] at (1150, 250, 200) mm
  - Disco_1175 [part] at (1250, 230, 200) mm
  - Placa_1176 [part] at (1150, 250, 200) mm
  - Placa_1177 [part] at (1150, 250, 200) mm
  - Placa_1178 [part] at (1150, 250, 200) mm
  - Disco_1179 [part] at (1250, 230, 200) mm
  - Disco_1180 [part] at (1250, 230, 200) mm
  - Disco_1181 [part] at (1250, 230, 200) mm
  - Disco_1182 [part] at (1250, 230, 200) mm
  - Placa_1183 [part] at (1150, 250, 200) mm
  - Placa_1184 [part] at (1150, 250, 200) mm
  - Disco_1185 [part] at (1250, 230, 200) mm
  - Disco_1186 [part] at (1250, 230, 200) mm
  - Disco_1187 [part] at (1250, 230, 200) mm
  - Placa_1188 [part] at (1150, 250, 200) mm
  - Disco_1189 [part] at (1250, 230, 200) mm
  - Disco_1190 [part] at (1250, 230, 200) mm
  - Disco_1191 [part] at (1250, 230, 200) mm
  - Disco_1192 [part] at (1250, 230, 200) mm
  - Disco_1193 [part] at (1250, 230, 200) mm
  - Placa_1194 [part] at (1150, 250, 200) mm
  - Disco_1195 [part] at (1250, 230, 200) mm
  - Disco_1196 [part] at (1250, 230, 200) mm
  - Placa_1197 [part] at (1146.4, 250, 200) mm
  - Placa_1198 [part] at (1150, 250, 200) mm
  - Disco_1199 [part] at (1250, 230, 200) mm
  - Disco_1200 [part] at (1250, 230, 200) mm
  - Disco_1201 [part] at (1250, 230, 200) mm
  - Disco_1202 [part] at (1250, 230, 200) mm
  - Placa_1203 [part] at (1150, 250, 200) mm
  - Disco_1204 [part] at (1250, 230, 200) mm
  - Placa_1205 [part] at (1150, 250, 200) mm
  - Placa_1206 [part] at (1150, 250, 200) mm
  - Disco_1207 [part] at (1250, 230, 200) mm
  - Placa_1208 [part] at (1150, 250, 200) mm
  - Disco_1209 [part] at (1250, 230, 200) mm
  - Disco_1210 [part] at (1250, 230, 200) mm
  - Placa_1211 [part] at (1150, 250, 200) mm
  - Disco_1212 [part] at (1250, 230, 200) mm
  - Placa_1213 [part] at (1150, 250, 200) mm
  - Disco_1214 [part] at (1250, 230, 200) mm
  - Placa_1215 [part] at (1150, 250, 200) mm
  - Placa_1216 [part] at (1150, 250, 200) mm
  - Disco_1217 [part] at (1250, 230, 200) mm
  - Placa_1218 [part] at (1150, 250, 200) mm
  - Disco_1219 [part] at (1250, 230, 200) mm
  - Placa_1220 [part] at (1150, 250, 200) mm
  - Placa_1221 [part] at (1150, 250, 200) mm
  - Disco_1222 [part] at (1250, 230, 200) mm
  - Disco_1223 [part] at (1250, 230, 200) mm
  - Placa_1224 [part] at (1150, 250, 200) mm
  - Placa_1225 [part] at (1150, 250, 200) mm
  - Placa_1226 [part] at (1150, 250, 200) mm
  - Placa_1227 [part] at (1150, 250, 200) mm
  - Disco_1228 [part] at (1250, 230, 200) mm
  - Disco_1229 [part] at (1250, 230, 200) mm
  - Disco_1230 [part] at (1250, 230, 200) mm
  - Placa_1231 [part] at (1150, 250, 200) mm
  - Disco_1232 [part] at (1250, 230, 200) mm
  - Placa_1233 [part] at (1150, 250, 200) mm
  - Placa_1234 [part] at (1150, 250, 200) mm
  - Placa_1235 [part] at (1150, 250, 200) mm
  - Disco_1236 [part] at (1250, 230, 200) mm
  - Disco_1237 [part] at (1250, 230, 200) mm
  - Placa_1238 [part] at (1150, 250, 200) mm
  - Disco_1239 [part] at (1250, 230, 200) mm
  - Placa_1240 [part] at (1150, 250, 200) mm
  - Placa_1241 [part] at (1150, 250, 200) mm
  - Placa_1242 [part] at (1150, 250, 200) mm
  - Disco_1243 [part] at (1250, 230, 200) mm
  - Disco_1244 [part] at (1250, 230, 200) mm
  - Disco_1245 [part] at (1250, 230, 200) mm
  - Placa_1246 [part] at (1146.4, 250, 200) mm
  - Disco_1247 [part] at (1250, 230, 200) mm
  - Placa_1248 [part] at (1150, 250, 200) mm
  - Placa_1249 [part] at (1150, 250, 200) mm
  - Disco_1250 [part] at (1250, 230, 200) mm
  - Placa_1251 [part] at (1150, 250, 200) mm
  - Disco_1252 [part] at (1250, 230, 200) mm
  - Disco_1253 [part] at (1250, 230, 200) mm
  - Disco_1254 [part] at (1250, 230, 200) mm
  - Placa_1255 [part] at (1150, 250, 200) mm
  - Placa_1256 [part] at (1150, 250, 200) mm
  - Disco_1257 [part] at (1250, 230, 200) mm
  - Disco_1258 [part] at (1250, 230, 200) mm
  - Disco_1259 [part] at (1250, 230, 200) mm
  - Placa_1260 [part] at (1150, 250, 200) mm
  - Disco_1261 [part] at (1250, 230, 200) mm
  - Placa_1262 [part] at (1150, 250, 200) mm
  - Disco_1263 [part] at (1250, 230, 200) mm
  - Disco_1264 [part] at (1250, 230, 200) mm
  - Disco_1265 [part] at (1250, 230, 200) mm
  - Placa_1266 [part] at (1150, 250, 200) mm
  - Placa_1267 [part] at (1150, 250, 200) mm
  - Disco_1268 [part] at (1250, 230, 200) mm
  - Disco_1269 [part] at (1250, 230, 200) mm
  - Placa_1270 [part] at (1150, 250, 200) mm
  - Placa_1271 [part] at (1150, 250, 200) mm
  - Placa_27 [part] at (1150, 250, 200) mm
  - Placa_28 [part] at (1150, 250, 200) mm
  - Placa_29 [part] at (1150, 250, 200) mm
  - Disco_30 [part] at (1250, 230, 200) mm
  - Disco_31 [part] at (1250, 230, 200) mm
  - Placa_32 [part] at (1150, 250, 200) mm
  - Placa_33 [part] at (1146.4, 250, 200) mm
  - Placa_34 [part] at (1150, 250, 200) mm
  - Disco_35 [part] at (1250, 230, 200) mm
  - Disco_36 [part] at (1250, 230, 200) mm
  - Disco_37 [part] at (1250, 230, 200) mm
  - Disco_38 [part] at (1250, 230, 200) mm
  - Placa_39 [part] at (1150, 250, 200) mm
  - Placa_40 [part] at (1150, 250, 200) mm
  - Placa_41 [part] at (1150, 250, 200) mm
  - Placa_42 [part] at (1150, 250, 200) mm
  - Disco_43 [part] at (1246.4, 230, 200) mm
  - Disco_44 [part] at (1250, 230, 200) mm
  - Disco_45 [part] at (1250, 230, 200) mm
  - Disco_46 [part] at (1250, 230, 200) mm
  - Placa_47 [part] at (1150, 250, 200) mm
  - Disco_48 [part] at (1250, 230, 200) mm
  - Placa_49 [part] at (1150, 250, 200) mm
  - Placa_50 [part] at (1150, 250, 200) mm
  - Disco_51 [part] at (1250, 230, 200) mm
  - Placa_52 [part] at (1150, 250, 200) mm
  - Disco_53 [part] at (1246.4, 230, 200) mm
  - Placa_54 [part] at (1150, 250, 200) mm
  - Placa_55 [part] at (1150, 250, 200) mm
  - Placa_56 [part] at (1150, 250, 200) mm
  - Disco_57 [part] at (1250, 230, 200) mm
  - Disco_58 [part] at (1250, 230, 200) mm
  - Placa_59 [part] at (1150, 250, 200) mm
  - Disco_60 [part] at (1250, 230, 200) mm
  - Placa_61 [part] at (1150, 250, 200) mm
  - Placa_62 [part] at (1150, 250, 200) mm
  - Disco_63 [part] at (1250, 230, 200) mm
  - Placa_64 [part] at (1150, 250, 200) mm
  - Disco_65 [part] at (1250, 230, 200) mm
  - Disco_66 [part] at (1250, 230, 200) mm
  - Disco_67 [part] at (1250, 230, 200) mm
  - Placa_68 [part] at (1150, 250, 200) mm
  - Placa_69 [part] at (1150, 250, 200) mm
  - Placa_70 [part] at (1150, 250, 200) mm
  - Placa_71 [part] at (1150, 250, 200) mm
  - Placa_72 [part] at (1150, 250, 200) mm
  - Placa_73 [part] at (1150, 250, 200) mm
  - Disco_74 [part] at (1250, 230, 200) mm
  - Disco_75 [part] at (1250, 230, 200) mm
  - Placa_76 [part] at (1150, 250, 200) mm
  - Disco_77 [part] at (1250, 230, 200) mm
  - Disco_78 [part] at (1250, 230, 200) mm
  - Disco_79 [part] at (1250, 230, 200) mm
  - Disco_80 [part] at (1250, 230, 200) mm
  - Placa_81 [part] at (1150, 250, 200) mm
  - Placa_82 [part] at (1150, 250, 200) mm
  - Placa_83 [part] at (1150, 250, 200) mm
  - Placa_84 [part] at (1150, 250, 200) mm
  - Disco_85 [part] at (1250, 230, 200) mm
  - Placa_86 [part] at (1150, 250, 200) mm
  - Disco_87 [part] at (1250, 230, 200) mm
  - Disco_88 [part] at (1250, 230, 200) mm
  - Placa_89 [part] at (1150, 250, 200) mm
  - Disco_90 [part] at (1250, 230, 200) mm
  - Disco_91 [part] at (1250, 230, 200) mm
  - Disco_92 [part] at (1250, 230, 200) mm
  - Placa_93 [part] at (1146.4, 250, 200) mm
  - Placa_94 [part] at (1150, 250, 200) mm
  - Disco_95 [part] at (1250, 230, 200) mm
  - Disco_96 [part] at (1250, 230, 200) mm
  - Disco_97 [part] at (1250, 230, 200) mm
  - Disco_98 [part] at (1250, 230, 200) mm
  - Disco_99 [part] at (1250, 230, 200) mm
  - Placa_100 [part] at (1150, 250, 200) mm
  - Placa_101 [part] at (1150, 250, 200) mm
  - Placa_102 [part] at (1150, 250, 200) mm
  - Disco_103 [part] at (1250, 230, 200) mm
  - Placa_104 [part] at (1150, 250, 200) mm
  - Disco_105 [part] at (1250, 230, 200) mm
  - Disco_106 [part] at (1250, 230, 200) mm
  - Placa_107 [part] at (1150, 250, 200) mm
  - Disco_108 [part] at (1250, 230, 200) mm
  - Disco_109 [part] at (1250, 230, 200) mm
  - Disco_110 [part] at (1250, 230, 200) mm
  - Placa_111 [part] at (1150, 250, 200) mm
  - Disco_112 [part] at (1250, 230, 200) mm
  - Disco_113 [part] at (1250, 230, 200) mm
  - Placa_114 [part] at (1146.4, 250, 200) mm
  - Disco_115 [part] at (1250, 230, 200) mm
  - Placa_116 [part] at (1150, 250, 200) mm
  - Placa_117 [part] at (1150, 250, 200) mm
  - Placa_118 [part] at (1150, 250, 200) mm
  - Placa_119 [part] at (1150, 250, 200) mm
  - Placa_120 [part] at (1150, 250, 200) mm
  - Placa_121 [part] at (1150, 250, 200) mm
  - Disco_122 [part] at (1250, 230, 200) mm
  - Placa_123 [part] at (1150, 250, 200) mm
  - Placa_124 [part] at (1146.4, 250, 200) mm
  - Placa_125 [part] at (1150, 250, 200) mm
  - Placa_126 [part] at (1150, 250, 200) mm
  - Disco_127 [part] at (1250, 230, 200) mm
  - Disco_128 [part] at (1250, 230, 200) mm
  - Disco_129 [part] at (1250, 230, 200) mm
  - Disco_130 [part] at (1250, 230, 200) mm
  - Placa_131 [part] at (1150, 250, 200) mm
  - Placa_132 [part] at (1150, 250, 200) mm
  - Placa_133 [part] at (1150, 250, 200) mm
  - Disco_134 [part] at (1246.4, 230, 200) mm
  - Placa_135 [part] at (1150, 250, 200) mm
  - Disco_136 [part] at (1250, 230, 200) mm
  - Placa_137 [part] at (1150, 250, 200) mm
  - Placa_138 [part] at (1150, 250, 200) mm
  - Disco_139 [part] at (1250, 230, 200) mm
  - Placa_140 [part] at (1150, 250, 200) mm
  - Placa_141 [part] at (1150, 250, 200) mm
  - Placa_142 [part] at (1150, 250, 200) mm
  - Placa_143 [part] at (1150, 250, 200) mm
  - Placa_144 [part] at (1146.4, 250, 200) mm
  - Placa_145 [part] at (1150, 250, 200) mm
  - Placa_146 [part] at (1150, 250, 200) mm
  - Disco_147 [part] at (1250, 230, 200) mm
  - Placa_148 [part] at (1150, 250, 200) mm
  - Disco_149 [part] at (1250, 230, 200) mm
  - Disco_150 [part] at (1250, 230, 200) mm
  - Placa_151 [part] at (1150, 250, 200) mm
  - Placa_152 [part] at (1150, 250, 200) mm
  - Placa_153 [part] at (1150, 250, 200) mm
  - Placa_154 [part] at (1150, 250, 200) mm
  - Disco_155 [part] at (1246.4, 230, 200) mm
  - Disco_156 [part] at (1250, 230, 200) mm
  - Placa_157 [part] at (1150, 250, 200) mm
  - Disco_158 [part] at (1250, 230, 200) mm
  - Disco_159 [part] at (1250, 230, 200) mm
  - Placa_160 [part] at (1150, 250, 200) mm
  - Disco_161 [part] at (1250, 230, 200) mm
  - Placa_162 [part] at (1150, 250, 200) mm
  - Disco_163 [part] at (1250, 230, 200) mm
  - Disco_164 [part] at (1250, 230, 200) mm
  - Disco_165 [part] at (1250, 230, 200) mm
  - Disco_166 [part] at (1246.4, 230, 200) mm
  - Disco_167 [part] at (1250, 230, 200) mm
  - Placa_168 [part] at (1150, 250, 200) mm
  - Disco_169 [part] at (1250, 230, 200) mm
  - Disco_170 [part] at (1250, 230, 200) mm
  - Disco_171 [part] at (1250, 230, 200) mm
  - Placa_172 [part] at (1150, 250, 200) mm
  - Disco_173 [part] at (1250, 230, 200) mm
  - Placa_174 [part] at (1150, 250, 200) mm
  - Placa_175 [part] at (1150, 250, 200) mm
  - Placa_176 [part] at (1146.4, 250, 200) mm
  - Placa_177 [part] at (1150, 250, 200) mm
  - Disco_178 [part] at (1250, 230, 200) mm
  - Disco_179 [part] at (1250, 230, 200) mm
  - Placa_180 [part] at (1150, 250, 200) mm
  - Placa_181 [part] at (1150, 250, 200) mm
  - Disco_182 [part] at (1250, 230, 200) mm
  - Disco_183 [part] at (1250, 230, 200) mm
  - Placa_184 [part] at (1150, 250, 200) mm
  - Placa_185 [part] at (1150, 250, 200) mm
  - Placa_186 [part] at (1146.4, 250, 200) mm
  - Placa_187 [part] at (1150, 250, 200) mm
  - Disco_188 [part] at (1250, 230, 200) mm
  - Disco_189 [part] at (1250, 230, 200) mm
  - Disco_190 [part] at (1250, 230, 200) mm
  - Placa_191 [part] at (1150, 250, 200) mm
  - Disco_192 [part] at (1250, 230, 200) mm
  - Disco_193 [part] at (1250, 230, 200) mm
  - Placa_194 [part] at (1150, 250, 200) mm
  - Placa_195 [part] at (1150, 250, 200) mm
  - Disco_196 [part] at (1246.4, 230, 200) mm
  - Placa_197 [part] at (1150, 250, 200) mm
  - Placa_198 [part] at (1150, 250, 200) mm
  - Disco_199 [part] at (1250, 230, 200) mm
  - Disco_200 [part] at (1250, 230, 200) mm
  - Disco_201 [part] at (1250, 230, 200) mm
  - Disco_202 [part] at (1250, 230, 200) mm
  - Placa_203 [part] at (1150, 250, 200) mm
  - Placa_204 [part] at (1150, 250, 200) mm
  - Disco_205 [part] at (1250, 230, 200) mm
  - Placa_206 [part] at (1150, 250, 200) mm
  - Disco_207 [part] at (1246.4, 230, 200) mm
  - Placa_208 [part] at (1150, 250, 200) mm
  - Placa_209 [part] at (1150, 250, 200) mm
  - Disco_210 [part] at (1250, 230, 200) mm
  - Placa_211 [part] at (1150, 250, 200) mm
  - Placa_212 [part] at (1150, 250, 200) mm
  - Disco_213 [part] at (1250, 230, 200) mm
  - Placa_214 [part] at (1150, 250, 200) mm
  - Disco_215 [part] at (1250, 230, 200) mm
  - Placa_216 [part] at (1150, 250, 200) mm
  - Disco_217 [part] at (1250, 230, 200) mm
  - Disco_218 [part] at (1246.4, 230, 200) mm
  - Disco_219 [part] at (1250, 230, 200) mm
  - Placa_220 [part] at (1150, 250, 200) mm
  - Disco_221 [part] at (1250, 230, 200) mm
  - Disco_222 [part] at (1250, 230, 200) mm
  - Placa_223 [part] at (1150, 250, 200) mm
  - Placa_224 [part] at (1150, 250, 200) mm
  - Placa_225 [part] at (1150, 250, 200) mm
  - Placa_226 [part] at (1150, 250, 200) mm
  - Disco_227 [part] at (1250, 230, 200) mm
  - Placa_228 [part] at (1150, 250, 200) mm
  - Disco_229 [part] at (1250, 230, 200) mm
  - Placa_230 [part] at (1150, 250, 200) mm
  - Disco_231 [part] at (1250, 230, 200) mm
  - Placa_232 [part] at (1150, 250, 200) mm
  - Placa_233 [part] at (1150, 250, 200) mm
  - Placa_234 [part] at (1150, 250, 200) mm
  - Disco_235 [part] at (1250, 230, 200) mm
  - Disco_236 [part] at (1250, 230, 200) mm
  - Placa_237 [part] at (1150, 250, 200) mm
  - Disco_238 [part] at (1250, 230, 200) mm
  - Placa_239 [part] at (1150, 250, 200) mm
  - Placa_240 [part] at (1150, 250, 200) mm
  - Placa_241 [part] at (1150, 250, 200) mm
  - Placa_242 [part] at (1150, 250, 200) mm
  - Disco_243 [part] at (1250, 230, 200) mm
  - Disco_244 [part] at (1250, 230, 200) mm
  - Placa_245 [part] at (1150, 250, 200) mm
  - Placa_246 [part] at (1150, 250, 200) mm
  - Placa_247 [part] at (1150, 250, 200) mm
  - Placa_248 [part] at (1150, 250, 200) mm
  - Disco_249 [part] at (1250, 230, 200) mm
  - Placa_250 [part] at (1150, 250, 200) mm
  - Placa_251 [part] at (1150, 250, 200) mm
  - Placa_252 [part] at (1150, 250, 200) mm
  - Disco_253 [part] at (1250, 230, 200) mm
  - Placa_254 [part] at (1150, 250, 200) mm
  - Disco_255 [part] at (1250, 230, 200) mm
  - Disco_256 [part] at (1250, 230, 200) mm
  - Placa_257 [part] at (1150, 250, 200) mm
  - Disco_258 [part] at (1250, 230, 200) mm
  - Disco_259 [part] at (1246.4, 230, 200) mm
  - Placa_260 [part] at (1150, 250, 200) mm
  - Disco_261 [part] at (1250, 230, 200) mm
  - Placa_262 [part] at (1150, 250, 200) mm
  - Placa_263 [part] at (1150, 250, 200) mm
  - Disco_264 [part] at (1250, 230, 200) mm
  - Disco_265 [part] at (1250, 230, 200) mm
  - Disco_266 [part] at (1250, 230, 200) mm
  - Disco_267 [part] at (1250, 230, 200) mm
  - Placa_268 [part] at (1150, 250, 200) mm
  - Disco_269 [part] at (1246.4, 230, 200) mm
  - Disco_270 [part] at (1250, 230, 200) mm
  - Disco_271 [part] at (1250, 230, 200) mm
  - Placa_272 [part] at (1150, 250, 200) mm
  - Placa_273 [part] at (1150, 250, 200) mm
  - Placa_274 [part] at (1150, 250, 200) mm
  - Disco_275 [part] at (1250, 230, 200) mm
  - Placa_276 [part] at (1150, 250, 200) mm
  - Placa_277 [part] at (1150, 250, 200) mm
  - Disco_278 [part] at (1250, 230, 200) mm
  - Placa_279 [part] at (1146.4, 250, 200) mm
  - Placa_280 [part] at (1150, 250, 200) mm
  - Placa_281 [part] at (1150, 250, 200) mm
  - Placa_282 [part] at (1150, 250, 200) mm
  - Disco_283 [part] at (1250, 230, 200) mm
  - Placa_284 [part] at (1150, 250, 200) mm
  - Placa_285 [part] at (1150, 250, 200) mm
  - Disco_286 [part] at (1250, 230, 200) mm
  - Disco_287 [part] at (1250, 230, 200) mm
  - Placa_288 [part] at (1150, 250, 200) mm
  - Disco_289 [part] at (1246.4, 230, 200) mm
  - Disco_290 [part] at (1250, 230, 200) mm
  - Disco_291 [part] at (1250, 230, 200) mm
  - Placa_292 [part] at (1150, 250, 200) mm
  - Disco_293 [part] at (1250, 230, 200) mm
  - Disco_294 [part] at (1250, 230, 200) mm
  - Placa_295 [part] at (1150, 250, 200) mm
  - Placa_296 [part] at (1150, 250, 200) mm
  - Disco_297 [part] at (1250, 230, 200) mm
  - Disco_298 [part] at (1250, 230, 200) mm
  - Disco_299 [part] at (1250, 230, 200) mm
  - Placa_300 [part] at (1146.4, 250, 200) mm
  - Placa_301 [part] at (1150, 250, 200) mm
  - Disco_302 [part] at (1250, 230, 200) mm
  - Disco_303 [part] at (1250, 230, 200) mm
  - Disco_304 [part] at (1250, 230, 200) mm
  - Disco_305 [part] at (1250, 230, 200) mm
  - Placa_306 [part] at (1150, 250, 200) mm
  - Placa_307 [part] at (1150, 250, 200) mm
  - Placa_308 [part] at (1150, 250, 200) mm
  - Placa_309 [part] at (1150, 250, 200) mm
  - Placa_310 [part] at (1150, 250, 200) mm
  - Disco_311 [part] at (1246.4, 230, 200) mm
  - Disco_312 [part] at (1250, 230, 200) mm
  - Disco_313 [part] at (1250, 230, 200) mm
  - Placa_314 [part] at (1150, 250, 200) mm
  - Placa_315 [part] at (1150, 250, 200) mm
  - Disco_316 [part] at (1250, 230, 200) mm
  - Placa_317 [part] at (1150, 250, 200) mm
  - Disco_318 [part] at (1250, 230, 200) mm
  - Placa_319 [part] at (1150, 250, 200) mm
  - Placa_320 [part] at (1150, 250, 200) mm
  - Placa_321 [part] at (1146.4, 250, 200) mm
  - Disco_322 [part] at (1250, 230, 200) mm
  - Disco_323 [part] at (1250, 230, 200) mm
  - Placa_324 [part] at (1150, 250, 200) mm
  - Placa_325 [part] at (1150, 250, 200) mm
  - Placa_326 [part] at (1150, 250, 200) mm
  - Placa_327 [part] at (1150, 250, 200) mm
  - Placa_328 [part] at (1150, 250, 200) mm
  - Placa_329 [part] at (1150, 250, 200) mm
  - Disco_330 [part] at (1250, 230, 200) mm
  - Disco_331 [part] at (1246.4, 230, 200) mm
  - Placa_332 [part] at (1150, 250, 200) mm
  - Disco_333 [part] at (1250, 230, 200) mm
  - Disco_334 [part] at (1250, 230, 200) mm
  - Placa_335 [part] at (1150, 250, 200) mm
  - Placa_336 [part] at (1150, 250, 200) mm
  - Disco_337 [part] at (1250, 230, 200) mm
  - Placa_338 [part] at (1150, 250, 200) mm
  - Disco_339 [part] at (1250, 230, 200) mm
  - Placa_340 [part] at (1150, 250, 200) mm
  - Disco_341 [part] at (1246.4, 230, 200) mm
  - Disco_342 [part] at (1250, 230, 200) mm
  - Placa_343 [part] at (1150, 250, 200) mm
  - Placa_344 [part] at (1150, 250, 200) mm
  - Disco_345 [part] at (1250, 230, 200) mm
  - Placa_346 [part] at (1150, 250, 200) mm
  - Disco_347 [part] at (1250, 230, 200) mm
  - Placa_348 [part] at (1150, 250, 200) mm
  - Disco_349 [part] at (1250, 230, 200) mm
  - Disco_350 [part] at (1250, 230, 200) mm
  - Placa_351 [part] at (1150, 250, 200) mm
  - Disco_352 [part] at (1246.4, 230, 200) mm
  - Disco_353 [part] at (1250, 230, 200) mm
  - Placa_354 [part] at (1150, 250, 200) mm
  - Placa_355 [part] at (1150, 250, 200) mm
  - Disco_356 [part] at (1250, 230, 200) mm
  - Placa_357 [part] at (1150, 250, 200) mm
  - Placa_358 [part] at (1150, 250, 200) mm
  - Placa_359 [part] at (1150, 250, 200) mm
  - Placa_360 [part] at (1150, 250, 200) mm
  - Disco_361 [part] at (1250, 230, 200) mm
  - Disco_362 [part] at (1250, 230, 200) mm
  - Placa_363 [part] at (1146.4, 250, 200) mm
  - Disco_364 [part] at (1250, 230, 200) mm
  - Disco_365 [part] at (1250, 230, 200) mm
  - Disco_366 [part] at (1250, 230, 200) mm
  - Disco_367 [part] at (1250, 230, 200) mm
  - Disco_368 [part] at (1250, 230, 200) mm
  - Placa_369 [part] at (1150, 250, 200) mm
  - Placa_370 [part] at (1150, 250, 200) mm
  - Placa_371 [part] at (1150, 250, 200) mm
  - Disco_372 [part] at (1250, 230, 200) mm
  - Placa_373 [part] at (1150, 250, 200) mm
  - Disco_374 [part] at (1250, 230, 200) mm
  - Disco_375 [part] at (1250, 230, 200) mm
  - Disco_376 [part] at (1250, 230, 200) mm
  - Placa_377 [part] at (1150, 250, 200) mm
  - Disco_378 [part] at (1250, 230, 200) mm
  - Placa_379 [part] at (1150, 250, 200) mm
  - Placa_380 [part] at (1150, 250, 200) mm
  - Disco_381 [part] at (1250, 230, 200) mm
  - Disco_382 [part] at (1250, 230, 200) mm
  - Disco_383 [part] at (1250, 230, 200) mm
  - Placa_384 [part] at (1150, 250, 200) mm
  - Disco_385 [part] at (1250, 230, 200) mm
  - Disco_386 [part] at (1250, 230, 200) mm
  - Disco_387 [part] at (1250, 230, 200) mm
  - Placa_388 [part] at (1150, 250, 200) mm
  - Disco_389 [part] at (1250, 230, 200) mm
  - Disco_390 [part] at (1250, 230, 200) mm
  - Disco_391 [part] at (1250, 230, 200) mm
  - Placa_392 [part] at (1150, 250, 200) mm
  - Placa_393 [part] at (1150, 250, 200) mm
  - Placa_394 [part] at (1150, 250, 200) mm
  - Disco_395 [part] at (1250, 230, 200) mm
  - Disco_396 [part] at (1250, 230, 200) mm
  - Placa_397 [part] at (1150, 250, 200) mm
  - Disco_398 [part] at (1250, 230, 200) mm
  - Placa_399 [part] at (1150, 250, 200) mm
  - Placa_400 [part] at (1150, 250, 200) mm
  - Placa_401 [part] at (1150, 250, 200) mm
  - Disco_402 [part] at (1250, 230, 200) mm
  - Placa_403 [part] at (1150, 250, 200) mm
  - Disco_404 [part] at (1250, 230, 200) mm
  - Placa_420 [part] at (1150, 250, 200) mm
  - Disco_421 [part] at (1250, 230, 200) mm
  - Placa_422 [part] at (1150, 250, 200) mm
  - Placa_423 [part] at (1150, 250, 200) mm
  - Placa_424 [part] at (1150, 250, 200) mm
  - Placa_425 [part] at (1150, 250, 200) mm
  - Disco_426 [part] at (1250, 230, 200) mm
  - Disco_427 [part] at (1250, 230, 200) mm
  - Disco_428 [part] at (1250, 230, 200) mm
  - Placa_429 [part] at (1150, 250, 200) mm
  - Disco_430 [part] at (1250, 230, 200) mm
  - Placa_431 [part] at (1150, 250, 200) mm
  - Disco_432 [part] at (1246.4, 230, 200) mm
  - Placa_433 [part] at (1150, 250, 200) mm
  - Disco_434 [part] at (1250, 230, 200) mm
  - Placa_435 [part] at (1150, 250, 200) mm
  - Placa_436 [part] at (1150, 250, 200) mm
  - Disco_437 [part] at (1250, 230, 200) mm
  - Placa_438 [part] at (1150, 250, 200) mm
  - Disco_439 [part] at (1250, 230, 200) mm
  - Placa_440 [part] at (1146.4, 250, 200) mm
  - Placa_441 [part] at (1150, 250, 200) mm
  - Placa_442 [part] at (1150, 250, 200) mm
  - Disco_443 [part] at (1250, 230, 200) mm
  - Placa_444 [part] at (1150, 250, 200) mm
  - Placa_445 [part] at (1150, 250, 200) mm
  - Disco_446 [part] at (1250, 230, 200) mm
  - Disco_447 [part] at (1250, 230, 200) mm
  - Placa_448 [part] at (1150, 250, 200) mm
  - Disco_449 [part] at (1246.4, 230, 200) mm
  - Disco_450 [part] at (1250, 230, 200) mm
  - Placa_451 [part] at (1150, 250, 200) mm
  - Placa_452 [part] at (1150, 250, 200) mm
  - Disco_453 [part] at (1250, 230, 200) mm
  - Placa_454 [part] at (1150, 250, 200) mm
  - Placa_455 [part] at (1150, 250, 200) mm
  - Disco_456 [part] at (1250, 230, 200) mm
  - Disco_457 [part] at (1250, 230, 200) mm
  - Disco_458 [part] at (1246.4, 230, 200) mm
  - Placa_459 [part] at (1150, 250, 200) mm
  - Disco_460 [part] at (1250, 230, 200) mm
  - Placa_461 [part] at (1150, 250, 200) mm
  - Disco_462 [part] at (1250, 230, 200) mm
  - Placa_463 [part] at (1150, 250, 200) mm
  - Disco_464 [part] at (1250, 230, 200) mm
  - Placa_465 [part] at (1150, 250, 200) mm
  - Disco_466 [part] at (1250, 230, 200) mm
  - Disco_467 [part] at (1246.4, 230, 200) mm
  - Placa_468 [part] at (1150, 250, 200) mm
  - Disco_469 [part] at (1250, 230, 200) mm
  - Disco_470 [part] at (1250, 230, 200) mm
  - Placa_471 [part] at (1150, 250, 200) mm
  - Disco_472 [part] at (1250, 230, 200) mm
  - Placa_473 [part] at (1150, 250, 200) mm
  - Placa_474 [part] at (1150, 250, 200) mm
  - Disco_475 [part] at (1250, 230, 200) mm
  - Disco_476 [part] at (1246.4, 230, 200) mm
  - Disco_477 [part] at (1250, 230, 200) mm
  - Disco_478 [part] at (1250, 230, 200) mm
  - Placa_479 [part] at (1150, 250, 200) mm
  - Placa_480 [part] at (1150, 250, 200) mm
  - Disco_481 [part] at (1250, 230, 200) mm
  - Placa_482 [part] at (1150, 250, 200) mm
  - Disco_483 [part] at (1250, 230, 200) mm
  - Disco_484 [part] at (1250, 230, 200) mm
  - Disco_485 [part] at (1246.4, 230, 200) mm
  - Disco_486 [part] at (1250, 230, 200) mm
  - Disco_487 [part] at (1250, 230, 200) mm
  - Placa_488 [part] at (1150, 250, 200) mm
  - Placa_489 [part] at (1150, 250, 200) mm
  - Placa_490 [part] at (1150, 250, 200) mm
  - Disco_491 [part] at (1250, 230, 200) mm
  - Disco_492 [part] at (1250, 230, 200) mm
  - Disco_493 [part] at (1250, 230, 200) mm
  - Disco_494 [part] at (1250, 230, 200) mm
  - Placa_495 [part] at (1150, 250, 200) mm
  - Placa_496 [part] at (1150, 250, 200) mm
  - Disco_497 [part] at (1250, 230, 200) mm
  - Placa_498 [part] at (1150, 250, 200) mm
  - Placa_499 [part] at (1150, 250, 200) mm
  - Disco_500 [part] at (1250, 230, 200) mm
  - Placa_501 [part] at (1150, 250, 200) mm
  - Disco_502 [part] at (1246.4, 230, 200) mm
  - Disco_503 [part] at (1250, 230, 200) mm
  - Placa_504 [part] at (1150, 250, 200) mm
  - Disco_505 [part] at (1250, 230, 200) mm
  - Disco_506 [part] at (1250, 230, 200) mm
  - Placa_507 [part] at (1150, 250, 200) mm
  - Placa_508 [part] at (1150, 250, 200) mm
  - Placa_509 [part] at (1150, 250, 200) mm
  - Disco_510 [part] at (1250, 230, 200) mm
  - Placa_511 [part] at (1146.4, 250, 200) mm
  - Disco_512 [part] at (1250, 230, 200) mm
  - Disco_513 [part] at (1250, 230, 200) mm
  - Disco_514 [part] at (1250, 230, 200) mm
  - Disco_515 [part] at (1250, 230, 200) mm
  - Placa_516 [part] at (1150, 250, 200) mm
  - Placa_517 [part] at (1150, 250, 200) mm
  - Disco_518 [part] at (1250, 230, 200) mm
  - Placa_519 [part] at (1150, 250, 200) mm
  - Placa_520 [part] at (1146.4, 250, 200) mm
  - Placa_521 [part] at (1150, 250, 200) mm
  - Placa_522 [part] at (1150, 250, 200) mm
  - Disco_523 [part] at (1250, 230, 200) mm
  - Disco_524 [part] at (1250, 230, 200) mm
  - Placa_525 [part] at (1150, 250, 200) mm
  - Placa_526 [part] at (1150, 250, 200) mm
  - Disco_527 [part] at (1250, 230, 200) mm
  - Disco_528 [part] at (1246.4, 230, 200) mm
  - Placa_529 [part] at (1150, 250, 200) mm
  - Disco_530 [part] at (1250, 230, 200) mm
  - Disco_531 [part] at (1250, 230, 200) mm
  - Placa_532 [part] at (1150, 250, 200) mm
  - Placa_533 [part] at (1150, 250, 200) mm
  - Disco_534 [part] at (1250, 230, 200) mm
  - Disco_535 [part] at (1250, 230, 200) mm
  - Placa_536 [part] at (1150, 250, 200) mm
  - Disco_537 [part] at (1246.4, 230, 200) mm
  - Disco_538 [part] at (1250, 230, 200) mm
  - Placa_539 [part] at (1150, 250, 200) mm
  - Disco_540 [part] at (1250, 230, 200) mm
  - Disco_541 [part] at (1250, 230, 200) mm
  - Placa_542 [part] at (1150, 250, 200) mm
  - Disco_543 [part] at (1250, 230, 200) mm
  - Disco_544 [part] at (1250, 230, 200) mm
  - Disco_545 [part] at (1250, 230, 200) mm
  - Disco_546 [part] at (1246.4, 230, 200) mm
  - Placa_547 [part] at (1150, 250, 200) mm
  - Placa_548 [part] at (1150, 250, 200) mm
  - Disco_549 [part] at (1250, 230, 200) mm
  - Disco_550 [part] at (1250, 230, 200) mm
  - Placa_551 [part] at (1150, 250, 200) mm
  - Placa_552 [part] at (1150, 250, 200) mm
  - Disco_553 [part] at (1250, 230, 200) mm
  - Placa_554 [part] at (1150, 250, 200) mm
  - Disco_555 [part] at (1246.4, 230, 200) mm
  - Disco_556 [part] at (1250, 230, 200) mm
  - Disco_557 [part] at (1250, 230, 200) mm
  - Placa_558 [part] at (1150, 250, 200) mm
  - Placa_559 [part] at (1150, 250, 200) mm
  - Placa_560 [part] at (1150, 250, 200) mm
  - Placa_561 [part] at (1150, 250, 200) mm
  - Disco_562 [part] at (1250, 230, 200) mm
  - Placa_563 [part] at (1146.4, 250, 200) mm
  - Disco_564 [part] at (1250, 230, 200) mm
  - Disco_565 [part] at (1250, 230, 200) mm
  - Disco_566 [part] at (1250, 230, 200) mm
  - Disco_567 [part] at (1250, 230, 200) mm
  - Disco_568 [part] at (1250, 230, 200) mm
  - Disco_569 [part] at (1250, 230, 200) mm
  - Disco_570 [part] at (1250, 230, 200) mm
  - Disco_571 [part] at (1250, 230, 200) mm
  - Placa_572 [part] at (1146.4, 250, 200) mm
  - Placa_573 [part] at (1150, 250, 200) mm
  - Placa_574 [part] at (1150, 250, 200) mm
  - Placa_575 [part] at (1150, 250, 200) mm
  - Disco_576 [part] at (1250, 230, 200) mm
  - Disco_577 [part] at (1250, 230, 200) mm
  - Placa_578 [part] at (1150, 250, 200) mm
  - Disco_579 [part] at (1250, 230, 200) mm
  - Placa_580 [part] at (1150, 250, 200) mm
  - Disco_581 [part] at (1246.4, 230, 200) mm
  - Disco_582 [part] at (1250, 230, 200) mm
  - Disco_583 [part] at (1250, 230, 200) mm
  - Placa_584 [part] at (1150, 250, 200) mm
  - Disco_585 [part] at (1250, 230, 200) mm
  - Disco_586 [part] at (1250, 230, 200) mm
  - Placa_587 [part] at (1150, 250, 200) mm
  - Placa_588 [part] at (1150, 250, 200) mm
  - Placa_589 [part] at (1150, 250, 200) mm
  - Placa_590 [part] at (1146.4, 250, 200) mm
  - Placa_591 [part] at (1150, 250, 200) mm
  - Disco_592 [part] at (1250, 230, 200) mm
  - Placa_593 [part] at (1150, 250, 200) mm
  - Disco_594 [part] at (1250, 230, 200) mm
  - Disco_595 [part] at (1250, 230, 200) mm
  - Placa_596 [part] at (1150, 250, 200) mm
  - Placa_597 [part] at (1150, 250, 200) mm
  - Disco_598 [part] at (1250, 230, 200) mm
  - Placa_599 [part] at (1146.4, 250, 200) mm
  - Disco_600 [part] at (1250, 230, 200) mm
  - Placa_601 [part] at (1150, 250, 200) mm
  - Placa_602 [part] at (1150, 250, 200) mm
  - Placa_603 [part] at (1150, 250, 200) mm
  - Placa_604 [part] at (1150, 250, 200) mm
  - Placa_605 [part] at (1150, 250, 200) mm
  - Disco_606 [part] at (1250, 230, 200) mm
  - Disco_607 [part] at (1250, 230, 200) mm
  - Disco_608 [part] at (1250, 230, 200) mm
  - Disco_609 [part] at (1250, 230, 200) mm
  - Disco_610 [part] at (1250, 230, 200) mm
  - Placa_611 [part] at (1150, 250, 200) mm
  - Disco_612 [part] at (1250, 230, 200) mm
  - Placa_613 [part] at (1150, 250, 200) mm
  - Disco_614 [part] at (1250, 230, 200) mm
  - Disco_615 [part] at (1250, 230, 200) mm
  - Disco_616 [part] at (1250, 230, 200) mm
  - Grupo_1 [graphiccomponentgroup]
    - Grupo_2 [graphiccomponentgroup]
  - Placa_4 [part] at (1146.4, 250, 200) mm
  - Disco_86 [part] at (1250, 230, 200) mm
  - Disco_87 [part] at (1250, 230, 200) mm
  - Placa_88 [part] at (1150, 250, 200) mm
  - Disco_89 [part] at (1250, 230, 200) mm
  - Placa_90 [part] at (1150, 250, 200) mm
  - Disco_91 [part] at (1246.4, 230, 200) mm
  - Placa_92 [part] at (1150, 250, 200) mm
  - Placa_93 [part] at (1150, 250, 200) mm
  - Placa_94 [part] at (1150, 250, 200) mm
  - Placa_95 [part] at (1150, 250, 200) mm
  - Placa_96 [part] at (1150, 250, 200) mm
  - Disco_97 [part] at (1250, 230, 200) mm
  - Disco_98 [part] at (1250, 230, 200) mm
  - Disco_99 [part] at (1246.4, 230, 200) mm
  - Placa_100 [part] at (1150, 250, 200) mm
  - Disco_101 [part] at (1250, 230, 200) mm
  - Disco_102 [part] at (1250, 230, 200) mm
  - Placa_103 [part] at (1150, 250, 200) mm
  - Disco_104 [part] at (1250, 230, 200) mm
  - Disco_105 [part] at (1250, 230, 200) mm
  - Placa_106 [part] at (1150, 250, 200) mm
  - Placa_107 [part] at (1146.4, 250, 200) mm
  - Disco_108 [part] at (1250, 230, 200) mm
  - Disco_109 [part] at (1250, 230, 200) mm
  - Disco_110 [part] at (1250, 230, 200) mm
  - Disco_111 [part] at (1250, 230, 200) mm
  - Placa_112 [part] at (1150, 250, 200) mm
  - Placa_113 [part] at (1150, 250, 200) mm
  - Disco_114 [part] at (1250, 230, 200) mm
  - Disco_115 [part] at (1246.4, 230, 200) mm
  - Placa_116 [part] at (1150, 250, 200) mm
  - Disco_117 [part] at (1250, 230, 200) mm
  - Disco_118 [part] at (1250, 230, 200) mm
  - Placa_119 [part] at (1150, 250, 200) mm
  - Disco_120 [part] at (1250, 230, 200) mm
  - Disco_121 [part] at (1250, 230, 200) mm
  - Disco_122 [part] at (1250, 230, 200) mm
  - Disco_123 [part] at (1246.4, 230, 200) mm
  - Placa_124 [part] at (1150, 250, 200) mm
  - Disco_125 [part] at (1250, 230, 200) mm
  - Placa_126 [part] at (1150, 250, 200) mm
  - Disco_127 [part] at (1250, 230, 200) mm
  - Disco_128 [part] at (1250, 230, 200) mm
  - Placa_129 [part] at (1150, 250, 200) mm
  - Disco_130 [part] at (1250, 230, 200) mm
  - Placa_131 [part] at (1146.4, 250, 200) mm
  - Disco_132 [part] at (1250, 230, 200) mm
  - Disco_133 [part] at (1250, 230, 200) mm
  - Disco_134 [part] at (1250, 230, 200) mm
  - Placa_135 [part] at (1150, 250, 200) mm
  - Placa_136 [part] at (1150, 250, 200) mm
  - Placa_137 [part] at (1150, 250, 200) mm
  - Disco_138 [part] at (1250, 230, 200) mm
  - Disco_139 [part] at (1250, 230, 200) mm
  - Disco_140 [part] at (1250, 230, 200) mm
  - Disco_141 [part] at (1250, 230, 200) mm
  - Disco_142 [part] at (1250, 230, 200) mm
  - Placa_143 [part] at (1150, 250, 200) mm
  - Disco_144 [part] at (1250, 230, 200) mm
  - Placa_145 [part] at (1150, 250, 200) mm
  - Disco_146 [part] at (1250, 230, 200) mm
  - Placa_147 [part] at (1146.4, 250, 200) mm
  - Disco_148 [part] at (1250, 230, 200) mm
  - Disco_149 [part] at (1250, 230, 200) mm
  - Placa_150 [part] at (1150, 250, 200) mm
  - Placa_151 [part] at (1150, 250, 200) mm
  - Disco_152 [part] at (1250, 230, 200) mm
  - Placa_153 [part] at (1150, 250, 200) mm
  - Disco_154 [part] at (1250, 230, 200) mm
  - Placa_155 [part] at (1146.4, 250, 200) mm
  - Disco_156 [part] at (1250, 230, 200) mm
  - Placa_157 [part] at (1150, 250, 200) mm
  - Placa_158 [part] at (1150, 250, 200) mm
  - Disco_159 [part] at (1250, 230, 200) mm
  - Disco_160 [part] at (1250, 230, 200) mm
  - Placa_161 [part] at (1150, 250, 200) mm
  - Placa_162 [part] at (1150, 250, 200) mm
  - Placa_163 [part] at (1146.4, 250, 200) mm
  - Placa_164 [part] at (1150, 250, 200) mm
  - Disco_165 [part] at (1250, 230, 200) mm
  - Placa_166 [part] at (1150, 250, 200) mm
  - Disco_167 [part] at (1250, 230, 200) mm
  - Placa_168 [part] at (1150, 250, 200) mm
  - Placa_169 [part] at (1150, 250, 200) mm
  - Placa_170 [part] at (1150, 250, 200) mm
  - Disco_171 [part] at (1250, 230, 200) mm
  - Placa_172 [part] at (1150, 250, 200) mm
  - Disco_173 [part] at (1250, 230, 200) mm
  - Disco_174 [part] at (1250, 230, 200) mm
